LIN {X 0,Y 368.877,Z 478.526,A -85,B 0,C 180,E1 -12822.01,E2 -12822.01} C_VEL
LIN {X 0,Y 368.882,Z 478.53,A -85,B 0,C 180,E1 -12825.178,E2 -12825.178} C_VEL
LIN {X 0,Y 368.881,Z 478.519,A -85,B 0,C 180,E1 -12828.179,E2 -12828.179} C_VEL
LIN {X 0,Y 368.909,Z 478.528,A -85,B 0,C 180,E1 -12831.36,E2 -12831.36} C_VEL
LIN {X 0,Y 368.935,Z 478.472,A -85,B 0,C 180,E1 -12835.147,E2 -12835.147} C_VEL
LIN {X 0,Y 368.929,Z 478.53,A -85,B 0,C 180,E1 -12839.047,E2 -12839.047} C_VEL
LIN {X 0,Y 368.963,Z 478.492,A -85,B 0,C 180,E1 -12842.797,E2 -12842.797} C_VEL
LIN {X 0,Y 368.946,Z 478.523,A -85,B 0,C 180,E1 -12846.113,E2 -12846.113} C_VEL
LIN {X 0,Y 368.935,Z 478.655,A -85,B 0,C 180,E1 -12848.554,E2 -12848.554} C_VEL
LIN {X 0,Y 369.153,Z 479.57,A -85,B 0,C 180,E1 -12848.747,E2 -12848.747} C_VEL
LIN {X 0,Y 377.34,Z 498.899,A -85,B 0,C 180,E1 -12849.662,E2 -12849.662} C_VEL
LIN {X 0,Y 376.778,Z 559.865,A -85,B 0,C 180,E1 -12850.864,E2 -12850.864} C_VEL
LIN {X 0,Y 376.605,Z 573.144,A -85,B 0,C 180,E1 -12851.334,E2 -12851.334} C_VEL
LIN {X 0,Y 376.21,Z 585.351,A -85,B 0,C 180,E1 -12851.978,E2 -12851.978} C_VEL
LIN {X 0,Y 375.597,Z 597.68,A -85,B 0,C 180,E1 -12852.858,E2 -12852.858} C_VEL
LIN {X 0,Y 374.644,Z 609.255,A -85,B 0,C 180,E1 -12853.937,E2 -12853.937} C_VEL
LIN {X 0,Y 373.753,Z 619.585,A -85,B 0,C 180,E1 -12855.156,E2 -12855.156} C_VEL
LIN {X 0,Y 372.946,Z 628.011,A -85,B 0,C 180,E1 -12856.376,E2 -12856.376} C_VEL
LIN {X 0,Y 372.21,Z 635.75,A -85,B 0,C 180,E1 -12857.736,E2 -12857.736} C_VEL
LIN {X 0,Y 371.314,Z 643.431,A -85,B 0,C 180,E1 -12859.393,E2 -12859.393} C_VEL
LIN {X 0,Y 370.669,Z 649.183,A -85,B 0,C 180,E1 -12860.944,E2 -12860.944} C_VEL
LIN {X 0,Y 370.256,Z 653.452,A -85,B 0,C 180,E1 -12862.365,E2 -12862.365} C_VEL
LIN {X 0,Y 369.654,Z 657.346,A -85,B 0,C 180,E1 -12863.998,E2 -12863.998} C_VEL
LIN {X 0,Y 369.252,Z 660.212,A -85,B 0,C 180,E1 -12865.634,E2 -12865.634} C_VEL
LIN {X 0,Y 369.235,Z 661.562,A -85,B 0,C 180,E1 -12866.727,E2 -12866.727} C_VEL
LIN {X 0,Y 369.048,Z 662.545,A -85,B 0,C 180,E1 -12867.817,E2 -12867.817} C_VEL
LIN {X 0,Y 369.11,Z 663.126,A -85,B 0,C 180,E1 -12868.909,E2 -12868.909} C_VEL
LIN {X 0,Y 369.091,Z 663.354,A -85,B 0,C 180,E1 -12870,E2 -12870} C_VEL
LIN {X 0,Y 369.11,Z 663.169,A -85,B 0,C 180,E1 -12871.091,E2 -12871.091} C_VEL
LIN {X 0,Y 369.048,Z 662.615,A -85,B 0,C 180,E1 -12872.183,E2 -12872.183} C_VEL
LIN {X 0,Y 369.232,Z 661.661,A -85,B 0,C 180,E1 -12873.273,E2 -12873.273} C_VEL
LIN {X 0,Y 369.243,Z 660.356,A -85,B 0,C 180,E1 -12874.366,E2 -12874.366} C_VEL
LIN {X 0,Y 369.647,Z 657.542,A -85,B 0,C 180,E1 -12876.002,E2 -12876.002} C_VEL
LIN {X 0,Y 370.232,Z 653.717,A -85,B 0,C 180,E1 -12877.636,E2 -12877.636} C_VEL
LIN {X 0,Y 370.699,Z 648.641,A -85,B 0,C 180,E1 -12879.328,E2 -12879.328} C_VEL
LIN {X 0,Y 371.431,Z 642.614,A -85,B 0,C 180,E1 -12880.907,E2 -12880.907} C_VEL
LIN {X 0,Y 372.346,Z 634.835,A -85,B 0,C 180,E1 -12882.536,E2 -12882.536} C_VEL
LIN {X 0,Y 373.257,Z 625.165,A -85,B 0,C 180,E1 -12884.168,E2 -12884.168} C_VEL
LIN {X 0,Y 374.143,Z 616.123,A -85,B 0,C 180,E1 -12885.386,E2 -12885.386} C_VEL
LIN {X 0,Y 375.038,Z 605.628,A -85,B 0,C 180,E1 -12886.528,E2 -12886.528} C_VEL
LIN {X 0,Y 375.806,Z 593.96,A -85,B 0,C 180,E1 -12887.536,E2 -12887.536} C_VEL
LIN {X 0,Y 376.424,Z 582.268,A -85,B 0,C 180,E1 -12888.308,E2 -12888.308} C_VEL
LIN {X 0,Y 376.764,Z 569.639,A -85,B 0,C 180,E1 -12888.911,E2 -12888.911} C_VEL
LIN {X 0,Y 376.825,Z 558.831,A -85,B 0,C 180,E1 -12889.261,E2 -12889.261} C_VEL
LIN {X 0,Y 376.782,Z 552.259,A -85,B 0,C 180,E1 -12889.408,E2 -12889.408} C_VEL
LIN {X 0,Y 376.155,Z 546.467,A -85,B 0,C 180,E1 -12889.559,E2 -12889.559} C_VEL
LIN {X 0,Y 371.059,Z 527.828,A -85,B 0,C 180,E1 -12890.233,E2 -12890.233} C_VEL
LIN {X 0,Y 370.516,Z 522.033,A -85,B 0,C 180,E1 -12890.383,E2 -12890.383} C_VEL
LIN {X 0,Y 370.808,Z 500.919,A -85,B 0,C 180,E1 -12890.796,E2 -12890.796} C_VEL
LIN {X 0,Y 362.693,Z 481.915,A -85,B 0,C 180,E1 -12891.708,E2 -12891.708} C_VEL
LIN {X 0,Y 361.991,Z 479.937,A -85,B 0,C 180,E1 -12891.87,E2 -12891.87} C_VEL
LIN {X 0,Y 361.91,Z 479.438,A -85,B 0,C 180,E1 -12892.1,E2 -12892.1} C_VEL
LIN {X 0,Y 361.929,Z 479.391,A -85,B 0,C 180,E1 -12895.289,E2 -12895.289} C_VEL
LIN {X 0,Y 361.908,Z 479.371,A -85,B 0,C 180,E1 -12897.778,E2 -12897.778} C_VEL
LIN {X 0,Y 361.837,Z 479.406,A -85,B 0,C 180,E1 -12901.629,E2 -12901.629} C_VEL
LIN {X 0,Y 361.873,Z 479.404,A -85,B 0,C 180,E1 -12905.344,E2 -12905.344} C_VEL
LIN {X 0,Y 361.869,Z 479.409,A -85,B 0,C 180,E1 -12909.026,E2 -12909.026} C_VEL
LIN {X 0,Y 361.833,Z 479.393,A -85,B 0,C 180,E1 -12912.828,E2 -12912.828} C_VEL
LIN {X 0,Y 361.832,Z 479.413,A -85,B 0,C 180,E1 -12915.943,E2 -12915.943} C_VEL
LIN {X 0,Y 361.83,Z 479.384,A -85,B 0,C 180,E1 -12919.244,E2 -12919.244} C_VEL
LIN {X 0,Y 361.859,Z 479.402,A -85,B 0,C 180,E1 -12922.776,E2 -12922.776} C_VEL
LIN {X 0,Y 361.849,Z 479.405,A -85,B 0,C 180,E1 -12925.719,E2 -12925.719} C_VEL
LIN {X 0,Y 361.871,Z 479.368,A -85,B 0,C 180,E1 -12929.672,E2 -12929.672} C_VEL
LIN {X 0,Y 361.949,Z 479.398,A -85,B 0,C 180,E1 -12933.474,E2 -12933.474} C_VEL
LIN {X 0,Y 361.883,Z 479.398,A -85,B 0,C 180,E1 -12937.144,E2 -12937.144} C_VEL
LIN {X 0,Y 361.899,Z 479.404,A -85,B 0,C 180,E1 -12940.723,E2 -12940.723} C_VEL
LIN {X 0,Y 361.925,Z 479.393,A -85,B 0,C 180,E1 -12943.066,E2 -12943.066} C_VEL
LIN {X 0,Y 361.991,Z 479.391,A -85,B 0,C 180,E1 -12946.527,E2 -12946.527} C_VEL
LIN {X 0,Y 362.024,Z 479.374,A -85,B 0,C 180,E1 -12949.938,E2 -12949.938} C_VEL
LIN {X 0,Y 362.143,Z 479.368,A -85,B 0,C 180,E1 -12952.192,E2 -12952.192} C_VEL
LIN {X 0,Y 362.11,Z 479.374,A -85,B 0,C 180,E1 -12954.431,E2 -12954.431} C_VEL
LIN {X 0,Y 362.275,Z 479.344,A -85,B 0,C 180,E1 -12957.776,E2 -12957.776} C_VEL
LIN {X 0,Y 362.421,Z 479.336,A -85,B 0,C 180,E1 -12960,E2 -12960} C_VEL
LIN {X 0,Y 362.275,Z 479.35,A -85,B 0,C 180,E1 -12962.224,E2 -12962.224} C_VEL
LIN {X 0,Y 362.16,Z 479.368,A -85,B 0,C 180,E1 -12966.686,E2 -12966.686} C_VEL
LIN {X 0,Y 362.023,Z 479.377,A -85,B 0,C 180,E1 -12970.062,E2 -12970.062} C_VEL
LIN {X 0,Y 361.99,Z 479.394,A -85,B 0,C 180,E1 -12973.899,E2 -12973.899} C_VEL
LIN {X 0,Y 361.96,Z 479.372,A -85,B 0,C 180,E1 -12977.939,E2 -12977.939} C_VEL
LIN {X 0,Y 361.876,Z 479.403,A -85,B 0,C 180,E1 -12981.654,E2 -12981.654} C_VEL
LIN {X 0,Y 361.921,Z 479.393,A -85,B 0,C 180,E1 -12985.291,E2 -12985.291} C_VEL
LIN {X 0,Y 361.917,Z 479.387,A -85,B 0,C 180,E1 -12987.778,E2 -12987.778} C_VEL
LIN {X 0,Y 361.841,Z 479.413,A -85,B 0,C 180,E1 -12991.286,E2 -12991.286} C_VEL
LIN {X 0,Y 361.849,Z 479.406,A -85,B 0,C 180,E1 -12994.281,E2 -12994.281} C_VEL
LIN {X 0,Y 361.86,Z 479.407,A -85,B 0,C 180,E1 -12997.224,E2 -12997.224} C_VEL
LIN {X 0,Y 361.832,Z 479.413,A -85,B 0,C 180,E1 -13000.756,E2 -13000.756} C_VEL
LIN {X 0,Y 361.842,Z 479.382,A -85,B 0,C 180,E1 -13004.365,E2 -13004.365} C_VEL
LIN {X 0,Y 361.881,Z 479.408,A -85,B 0,C 180,E1 -13007.561,E2 -13007.561} C_VEL
LIN {X 0,Y 361.872,Z 479.401,A -85,B 0,C 180,E1 -13010.973,E2 -13010.973} C_VEL
LIN {X 0,Y 361.906,Z 479.544,A -85,B 0,C 180,E1 -13014.756,E2 -13014.756} C_VEL
LIN {X 0,Y 365.118,Z 492.779,A -85,B 0,C 180,E1 -13017.591,E2 -13017.591} C_VEL
LIN {X 0,Y 367.943,Z 505.89,A -85,B 0,C 180,E1 -13020.224,E2 -13020.224} C_VEL
LIN {X 0,Y 367.28,Z 514.74,A -85,B 0,C 180,E1 -13021.796,E2 -13021.796} C_VEL
LIN {X 0,Y 364.961,Z 539.488,A -85,B 0,C 180,E1 -13026.148,E2 -13026.148} C_VEL
LIN {X 0,Y 364.188,Z 549.23,A -85,B 0,C 180,E1 -13027.834,E2 -13027.834} C_VEL
LIN {X 0,Y 368.3,Z 584.784,A -85,B 0,C 180,E1 -13028.832,E2 -13028.832} C_VEL
LIN {X 0,Y 369.534,Z 599.506,A -85,B 0,C 180,E1 -13029.201,E2 -13029.201} C_VEL
LIN {X 0,Y 368.537,Z 660.016,A -85,B 0,C 180,E1 -13030.397,E2 -13030.397} C_VEL
LIN {X 0,Y 367.865,Z 673.29,A -85,B 0,C 180,E1 -13030.867,E2 -13030.867} C_VEL
LIN {X 0,Y 366.915,Z 685.485,A -85,B 0,C 180,E1 -13031.504,E2 -13031.504} C_VEL
LIN {X 0,Y 365.68,Z 697.816,A -85,B 0,C 180,E1 -13032.381,E2 -13032.381} C_VEL
LIN {X 0,Y 364.603,Z 709.538,A -85,B 0,C 180,E1 -13033.482,E2 -13033.482} C_VEL
LIN {X 0,Y 363.558,Z 719.018,A -85,B 0,C 180,E1 -13034.586,E2 -13034.586} C_VEL
LIN {X 0,Y 362.501,Z 728.498,A -85,B 0,C 180,E1 -13035.932,E2 -13035.932} C_VEL
LIN {X 0,Y 362.19,Z 733.797,A -85,B 0,C 180,E1 -13036.821,E2 -13036.821} C_VEL
LIN {X 0,Y 361.524,Z 740.995,A -85,B 0,C 180,E1 -13038.222,E2 -13038.222} C_VEL
LIN {X 0,Y 361.08,Z 748.089,A -85,B 0,C 180,E1 -13039.911,E2 -13039.911} C_VEL
LIN {X 0,Y 360.92,Z 753.811,A -85,B 0,C 180,E1 -13041.603,E2 -13041.603} C_VEL
LIN {X 0,Y 360.946,Z 758.327,A -85,B 0,C 180,E1 -13043.291,E2 -13043.291} C_VEL
LIN {X 0,Y 361.025,Z 760.727,A -85,B 0,C 180,E1 -13044.414,E2 -13044.414} C_VEL
LIN {X 0,Y 361.182,Z 762.687,A -85,B 0,C 180,E1 -13045.536,E2 -13045.536} C_VEL
LIN {X 0,Y 361.271,Z 764.153,A -85,B 0,C 180,E1 -13046.654,E2 -13046.654} C_VEL
LIN {X 0,Y 361.67,Z 765.879,A -85,B 0,C 180,E1 -13048.887,E2 -13048.887} C_VEL
LIN {X 0,Y 361.734,Z 766.112,A -85,B 0,C 180,E1 -13050,E2 -13050} C_VEL
LIN {X 0,Y 361.67,Z 765.876,A -85,B 0,C 180,E1 -13051.113,E2 -13051.113} C_VEL
LIN {X 0,Y 361.274,Z 764.148,A -85,B 0,C 180,E1 -13053.346,E2 -13053.346} C_VEL
LIN {X 0,Y 361.19,Z 762.678,A -85,B 0,C 180,E1 -13054.464,E2 -13054.464} C_VEL
LIN {X 0,Y 361.019,Z 759.595,A -85,B 0,C 180,E1 -13056.146,E2 -13056.146} C_VEL
LIN {X 0,Y 360.914,Z 755.441,A -85,B 0,C 180,E1 -13057.834,E2 -13057.834} C_VEL
LIN {X 0,Y 361.055,Z 749.1,A -85,B 0,C 180,E1 -13059.806,E2 -13059.806} C_VEL
LIN {X 0,Y 361.453,Z 742.222,A -85,B 0,C 180,E1 -13061.496,E2 -13061.496} C_VEL
LIN {X 0,Y 362.184,Z 733.742,A -85,B 0,C 180,E1 -13063.179,E2 -13063.179} C_VEL
LIN {X 0,Y 362.895,Z 725.06,A -85,B 0,C 180,E1 -13064.582,E2 -13064.582} C_VEL
LIN {X 0,Y 363.82,Z 715.587,A -85,B 0,C 180,E1 -13065.834,E2 -13065.834} C_VEL
LIN {X 0,Y 365.095,Z 703.902,A -85,B 0,C 180,E1 -13067.071,E2 -13067.071} C_VEL
LIN {X 0,Y 366.265,Z 692.423,A -85,B 0,C 180,E1 -13068.023,E2 -13068.023} C_VEL
LIN {X 0,Y 367.281,Z 680.646,A -85,B 0,C 180,E1 -13068.766,E2 -13068.766} C_VEL
LIN {X 0,Y 368.186,Z 667.106,A -85,B 0,C 180,E1 -13069.369,E2 -13069.369} C_VEL
LIN {X 0,Y 368.651,Z 653.646,A -85,B 0,C 180,E1 -13069.742,E2 -13069.742} C_VEL
LIN {X 0,Y 369.378,Z 596.606,A -85,B 0,C 180,E1 -13070.854,E2 -13070.854} C_VEL
LIN {X 0,Y 365.691,Z 561.697,A -85,B 0,C 180,E1 -13071.779,E2 -13071.779} C_VEL
LIN {X 0,Y 364.181,Z 549.137,A -85,B 0,C 180,E1 -13072.162,E2 -13072.162} C_VEL
LIN {X 0,Y 366.138,Z 526.073,A -85,B 0,C 180,E1 -13076.198,E2 -13076.198} C_VEL
LIN {X 0,Y 367.987,Z 507.54,A -85,B 0,C 180,E1 -13079.457,E2 -13079.457} C_VEL
LIN {X 0,Y 367.443,Z 503.107,A -85,B 0,C 180,E1 -13080.304,E2 -13080.304} C_VEL
LIN {X 0,Y 363.861,Z 487.384,A -85,B 0,C 180,E1 -13083.515,E2 -13083.515} C_VEL
LIN {X 0,Y 361.898,Z 479.519,A -85,B 0,C 180,E1 -13085.245,E2 -13085.245} C_VEL
LIN {X 0,Y 361.872,Z 479.401,A -85,B 0,C 180,E1 -13089.027,E2 -13089.027} C_VEL
LIN {X 0,Y 361.881,Z 479.409,A -85,B 0,C 180,E1 -13092.439,E2 -13092.439} C_VEL
LIN {X 0,Y 361.842,Z 479.382,A -85,B 0,C 180,E1 -13095.635,E2 -13095.635} C_VEL
LIN {X 0,Y 361.832,Z 479.412,A -85,B 0,C 180,E1 -13099.244,E2 -13099.244} C_VEL
LIN {X 0,Y 361.86,Z 479.407,A -85,B 0,C 180,E1 -13102.776,E2 -13102.776} C_VEL
LIN {X 0,Y 361.849,Z 479.405,A -85,B 0,C 180,E1 -13105.719,E2 -13105.719} C_VEL
LIN {X 0,Y 361.872,Z 479.408,A -85,B 0,C 180,E1 -13109.672,E2 -13109.672} C_VEL
LIN {X 0,Y 361.948,Z 479.378,A -85,B 0,C 180,E1 -13113.475,E2 -13113.475} C_VEL
LIN {X 0,Y 361.883,Z 479.405,A -85,B 0,C 180,E1 -13117.144,E2 -13117.144} C_VEL
LIN {X 0,Y 361.881,Z 479.38,A -85,B 0,C 180,E1 -13120.722,E2 -13120.722} C_VEL
LIN {X 0,Y 361.925,Z 479.393,A -85,B 0,C 180,E1 -13123.066,E2 -13123.066} C_VEL
LIN {X 0,Y 361.991,Z 479.393,A -85,B 0,C 180,E1 -13126.528,E2 -13126.528} C_VEL
LIN {X 0,Y 362.023,Z 479.378,A -85,B 0,C 180,E1 -13129.938,E2 -13129.938} C_VEL
LIN {X 0,Y 362.16,Z 479.368,A -85,B 0,C 180,E1 -13133.314,E2 -13133.314} C_VEL
LIN {X 0,Y 362.275,Z 479.353,A -85,B 0,C 180,E1 -13137.776,E2 -13137.776} C_VEL
LIN {X 0,Y 362.421,Z 479.338,A -85,B 0,C 180,E1 -13140,E2 -13140} C_VEL
LIN {X 0,Y 362.275,Z 479.346,A -85,B 0,C 180,E1 -13142.224,E2 -13142.224} C_VEL
LIN {X 0,Y 362.16,Z 479.372,A -85,B 0,C 180,E1 -13146.686,E2 -13146.686} C_VEL
LIN {X 0,Y 362.024,Z 479.374,A -85,B 0,C 180,E1 -13150.062,E2 -13150.062} C_VEL
LIN {X 0,Y 361.99,Z 479.39,A -85,B 0,C 180,E1 -13153.899,E2 -13153.899} C_VEL
LIN {X 0,Y 361.96,Z 479.392,A -85,B 0,C 180,E1 -13157.939,E2 -13157.939} C_VEL
LIN {X 0,Y 361.876,Z 479.397,A -85,B 0,C 180,E1 -13161.654,E2 -13161.654} C_VEL
LIN {X 0,Y 361.922,Z 479.402,A -85,B 0,C 180,E1 -13165.291,E2 -13165.291} C_VEL
LIN {X 0,Y 361.916,Z 479.391,A -85,B 0,C 180,E1 -13167.779,E2 -13167.779} C_VEL
LIN {X 0,Y 361.841,Z 479.373,A -85,B 0,C 180,E1 -13171.286,E2 -13171.286} C_VEL
LIN {X 0,Y 361.849,Z 479.404,A -85,B 0,C 180,E1 -13174.281,E2 -13174.281} C_VEL
LIN {X 0,Y 361.859,Z 479.403,A -85,B 0,C 180,E1 -13177.224,E2 -13177.224} C_VEL
LIN {X 0,Y 361.83,Z 479.384,A -85,B 0,C 180,E1 -13180.756,E2 -13180.756} C_VEL
LIN {X 0,Y 361.843,Z 479.412,A -85,B 0,C 180,E1 -13184.365,E2 -13184.365} C_VEL
LIN {X 0,Y 361.834,Z 479.392,A -85,B 0,C 180,E1 -13187.569,E2 -13187.569} C_VEL
LIN {X 0,Y 361.87,Z 479.409,A -85,B 0,C 180,E1 -13190.974,E2 -13190.974} C_VEL
LIN {X 0,Y 361.873,Z 479.354,A -85,B 0,C 180,E1 -13194.656,E2 -13194.656} C_VEL
LIN {X 0,Y 361.837,Z 479.405,A -85,B 0,C 180,E1 -13198.371,E2 -13198.371} C_VEL
LIN {X 0,Y 361.908,Z 479.373,A -85,B 0,C 180,E1 -13202.222,E2 -13202.222} C_VEL
LIN {X 0,Y 361.929,Z 479.389,A -85,B 0,C 180,E1 -13204.711,E2 -13204.711} C_VEL
LIN {X 0,Y 361.913,Z 479.54,A -85,B 0,C 180,E1 -13208.124,E2 -13208.124} C_VEL
LIN {X 0,Y 362.139,Z 480.575,A -85,B 0,C 180,E1 -13208.317,E2 -13208.317} C_VEL
LIN {X 0,Y 370.357,Z 499.721,A -85,B 0,C 180,E1 -13209.256,E2 -13209.256} C_VEL
LIN {X 0,Y 370.821,Z 501.605,A -85,B 0,C 180,E1 -13209.323,E2 -13209.323} C_VEL
LIN {X 0,Y 370.139,Z 559.915,A -85,B 0,C 180,E1 -13210.484,E2 -13210.484} C_VEL
LIN {X 0,Y 369.975,Z 572.765,A -85,B 0,C 180,E1 -13210.921,E2 -13210.921} C_VEL
LIN {X 0,Y 369.575,Z 585.231,A -85,B 0,C 180,E1 -13211.571,E2 -13211.571} C_VEL
LIN {X 0,Y 368.939,Z 597.581,A -85,B 0,C 180,E1 -13212.448,E2 -13212.448} C_VEL
LIN {X 0,Y 368.008,Z 608.977,A -85,B 0,C 180,E1 -13213.497,E2 -13213.497} C_VEL
LIN {X 0,Y 367.031,Z 619.532,A -85,B 0,C 180,E1 -13214.735,E2 -13214.735} C_VEL
LIN {X 0,Y 366.119,Z 629.002,A -85,B 0,C 180,E1 -13216.117,E2 -13216.117} C_VEL
LIN {X 0,Y 365.345,Z 636.74,A -85,B 0,C 180,E1 -13217.502,E2 -13217.502} C_VEL
LIN {X 0,Y 364.409,Z 644.421,A -85,B 0,C 180,E1 -13219.19,E2 -13219.19} C_VEL
LIN {X 0,Y 363.73,Z 650.173,A -85,B 0,C 180,E1 -13220.77,E2 -13220.77} C_VEL
LIN {X 0,Y 363.292,Z 654.441,A -85,B 0,C 180,E1 -13222.217,E2 -13222.217} C_VEL
LIN {X 0,Y 362.665,Z 658.335,A -85,B 0,C 180,E1 -13223.882,E2 -13223.882} C_VEL
LIN {X 0,Y 362.243,Z 661.202,A -85,B 0,C 180,E1 -13225.549,E2 -13225.549} C_VEL
LIN {X 0,Y 362.218,Z 662.551,A -85,B 0,C 180,E1 -13226.663,E2 -13226.663} C_VEL
LIN {X 0,Y 362.027,Z 663.533,A -85,B 0,C 180,E1 -13227.775,E2 -13227.775} C_VEL
LIN {X 0,Y 362.085,Z 664.114,A -85,B 0,C 180,E1 -13228.888,E2 -13228.888} C_VEL
LIN {X 0,Y 362.065,Z 664.342,A -85,B 0,C 180,E1 -13230,E2 -13230} C_VEL
LIN {X 0,Y 362.085,Z 664.156,A -85,B 0,C 180,E1 -13231.112,E2 -13231.112} C_VEL
LIN {X 0,Y 362.026,Z 663.603,A -85,B 0,C 180,E1 -13232.225,E2 -13232.225} C_VEL
LIN {X 0,Y 362.215,Z 662.648,A -85,B 0,C 180,E1 -13233.337,E2 -13233.337} C_VEL
LIN {X 0,Y 362.232,Z 661.344,A -85,B 0,C 180,E1 -13234.451,E2 -13234.451} C_VEL
LIN {X 0,Y 362.657,Z 658.53,A -85,B 0,C 180,E1 -13236.118,E2 -13236.118} C_VEL
LIN {X 0,Y 363.268,Z 654.704,A -85,B 0,C 180,E1 -13237.783,E2 -13237.783} C_VEL
LIN {X 0,Y 363.765,Z 649.628,A -85,B 0,C 180,E1 -13239.508,E2 -13239.508} C_VEL
LIN {X 0,Y 364.532,Z 643.6,A -85,B 0,C 180,E1 -13241.116,E2 -13241.116} C_VEL
LIN {X 0,Y 365.488,Z 635.821,A -85,B 0,C 180,E1 -13242.775,E2 -13242.775} C_VEL
LIN {X 0,Y 366.445,Z 626.151,A -85,B 0,C 180,E1 -13244.437,E2 -13244.437} C_VEL
LIN {X 0,Y 367.355,Z 617.11,A -85,B 0,C 180,E1 -13245.678,E2 -13245.678} C_VEL
LIN {X 0,Y 368.301,Z 606.613,A -85,B 0,C 180,E1 -13246.839,E2 -13246.839} C_VEL
LIN {X 0,Y 369.089,Z 595.098,A -85,B 0,C 180,E1 -13247.853,E2 -13247.853} C_VEL
LIN {X 0,Y 369.752,Z 583.832,A -85,B 0,C 180,E1 -13248.614,E2 -13248.614} C_VEL
LIN {X 0,Y 370.09,Z 571.524,A -85,B 0,C 180,E1 -13249.229,E2 -13249.229} C_VEL
LIN {X 0,Y 370.196,Z 559.798,A -85,B 0,C 180,E1 -13249.62,E2 -13249.62} C_VEL
LIN {X 0,Y 370.506,Z 523.206,A -85,B 0,C 180,E1 -13250.36,E2 -13250.36} C_VEL
LIN {X 0,Y 370.516,Z 522.033,A -85,B 0,C 180,E1 -13250.383,E2 -13250.383} C_VEL
LIN {X 0,Y 369.893,Z 516.227,A -85,B 0,C 180,E1 -13250.54,E2 -13250.54} C_VEL
LIN {X 0,Y 368.235,Z 510.668,A -85,B 0,C 180,E1 -13250.756,E2 -13250.756} C_VEL
LIN {X 0,Y 360.193,Z 492.917,A -85,B 0,C 180,E1 -13251.641,E2 -13251.641} C_VEL
LIN {X 0,Y 355.081,Z 481.33,A -85,B 0,C 180,E1 -13252.256,E2 -13252.256} C_VEL
LIN {X 0,Y 354.878,Z 480.41,A -85,B 0,C 180,E1 -13252.462,E2 -13252.462} C_VEL
LIN {X 0,Y 354.9,Z 480.253,A -85,B 0,C 180,E1 -13255.827,E2 -13255.827} C_VEL
LIN {X 0,Y 354.817,Z 480.284,A -85,B 0,C 180,E1 -13259.681,E2 -13259.681} C_VEL
LIN {X 0,Y 354.805,Z 480.288,A -85,B 0,C 180,E1 -13263.701,E2 -13263.701} C_VEL
LIN {X 0,Y 354.797,Z 480.277,A -85,B 0,C 180,E1 -13266.459,E2 -13266.459} C_VEL
LIN {X 0,Y 354.822,Z 480.289,A -85,B 0,C 180,E1 -13269.423,E2 -13269.423} C_VEL
LIN {X 0,Y 354.785,Z 480.27,A -85,B 0,C 180,E1 -13272.866,E2 -13272.866} C_VEL
LIN {X 0,Y 354.778,Z 480.292,A -85,B 0,C 180,E1 -13276.105,E2 -13276.105} C_VEL
LIN {X 0,Y 354.783,Z 480.262,A -85,B 0,C 180,E1 -13279.178,E2 -13279.178} C_VEL
LIN {X 0,Y 354.803,Z 480.279,A -85,B 0,C 180,E1 -13282.402,E2 -13282.402} C_VEL
LIN {X 0,Y 354.808,Z 480.291,A -85,B 0,C 180,E1 -13284.94,E2 -13284.94} C_VEL
LIN {X 0,Y 354.788,Z 480.254,A -85,B 0,C 180,E1 -13288.404,E2 -13288.404} C_VEL
LIN {X 0,Y 354.848,Z 480.263,A -85,B 0,C 180,E1 -13291.619,E2 -13291.619} C_VEL
LIN {X 0,Y 354.893,Z 480.275,A -85,B 0,C 180,E1 -13294.172,E2 -13294.172} C_VEL
LIN {X 0,Y 354.823,Z 480.275,A -85,B 0,C 180,E1 -13297.893,E2 -13297.893} C_VEL
LIN {X 0,Y 354.915,Z 480.27,A -85,B 0,C 180,E1 -13301.891,E2 -13301.891} C_VEL
LIN {X 0,Y 354.935,Z 480.27,A -85,B 0,C 180,E1 -13305.981,E2 -13305.981} C_VEL
LIN {X 0,Y 354.97,Z 480.253,A -85,B 0,C 180,E1 -13309.736,E2 -13309.736} C_VEL
LIN {X 0,Y 355.106,Z 480.245,A -85,B 0,C 180,E1 -13312.037,E2 -13312.037} C_VEL
LIN {X 0,Y 355.084,Z 480.249,A -85,B 0,C 180,E1 -13314.32,E2 -13314.32} C_VEL
LIN {X 0,Y 355.238,Z 480.22,A -85,B 0,C 180,E1 -13317.732,E2 -13317.732} C_VEL
LIN {X 0,Y 355.391,Z 480.212,A -85,B 0,C 180,E1 -13320,E2 -13320} C_VEL
LIN {X 0,Y 355.238,Z 480.226,A -85,B 0,C 180,E1 -13322.268,E2 -13322.268} C_VEL
LIN {X 0,Y 355.122,Z 480.245,A -85,B 0,C 180,E1 -13326.819,E2 -13326.819} C_VEL
LIN {X 0,Y 354.97,Z 480.254,A -85,B 0,C 180,E1 -13330.264,E2 -13330.264} C_VEL
LIN {X 0,Y 354.935,Z 480.272,A -85,B 0,C 180,E1 -13334.019,E2 -13334.019} C_VEL
LIN {X 0,Y 354.915,Z 480.248,A -85,B 0,C 180,E1 -13338.109,E2 -13338.109} C_VEL
LIN {X 0,Y 354.823,Z 480.286,A -85,B 0,C 180,E1 -13342.107,E2 -13342.107} C_VEL
LIN {X 0,Y 354.893,Z 480.26,A -85,B 0,C 180,E1 -13345.828,E2 -13345.828} C_VEL
LIN {X 0,Y 354.849,Z 480.284,A -85,B 0,C 180,E1 -13349.679,E2 -13349.679} C_VEL
LIN {X 0,Y 354.801,Z 480.276,A -85,B 0,C 180,E1 -13353.703,E2 -13353.703} C_VEL
LIN {X 0,Y 354.793,Z 480.288,A -85,B 0,C 180,E1 -13356.46,E2 -13356.46} C_VEL
LIN {X 0,Y 354.82,Z 480.283,A -85,B 0,C 180,E1 -13359.424,E2 -13359.424} C_VEL
LIN {X 0,Y 354.786,Z 480.268,A -85,B 0,C 180,E1 -13362.868,E2 -13362.868} C_VEL
LIN {X 0,Y 354.849,Z 480.277,A -85,B 0,C 180,E1 -13366.118,E2 -13366.118} C_VEL
LIN {X 0,Y 354.853,Z 480.264,A -85,B 0,C 180,E1 -13369.189,E2 -13369.189} C_VEL
LIN {X 0,Y 354.807,Z 480.284,A -85,B 0,C 180,E1 -13372.403,E2 -13372.403} C_VEL
LIN {X 0,Y 354.863,Z 480.538,A -85,B 0,C 180,E1 -13374.363,E2 -13374.363} C_VEL
LIN {X 0,Y 358.004,Z 493.339,A -85,B 0,C 180,E1 -13377.169,E2 -13377.169} C_VEL
LIN {X 0,Y 360.932,Z 506.614,A -85,B 0,C 180,E1 -13379.908,E2 -13379.908} C_VEL
LIN {X 0,Y 360.973,Z 510.056,A -85,B 0,C 180,E1 -13380.555,E2 -13380.555} C_VEL
LIN {X 0,Y 358.83,Z 530.823,A -85,B 0,C 180,E1 -13384.284,E2 -13384.284} C_VEL
LIN {X 0,Y 357.342,Z 548.301,A -85,B 0,C 180,E1 -13387.392,E2 -13387.392} C_VEL
LIN {X 0,Y 361.535,Z 584.354,A -85,B 0,C 180,E1 -13388.428,E2 -13388.428} C_VEL
LIN {X 0,Y 362.817,Z 600.626,A -85,B 0,C 180,E1 -13388.841,E2 -13388.841} C_VEL
LIN {X 0,Y 361.821,Z 659.025,A -85,B 0,C 180,E1 -13390.018,E2 -13390.018} C_VEL
LIN {X 0,Y 361.137,Z 672.296,A -85,B 0,C 180,E1 -13390.496,E2 -13390.496} C_VEL
LIN {X 0,Y 360.142,Z 684.486,A -85,B 0,C 180,E1 -13391.143,E2 -13391.143} C_VEL
LIN {X 0,Y 358.907,Z 696.821,A -85,B 0,C 180,E1 -13392.037,E2 -13392.037} C_VEL
LIN {X 0,Y 357.72,Z 708.531,A -85,B 0,C 180,E1 -13393.155,E2 -13393.155} C_VEL
LIN {X 0,Y 356.643,Z 718.012,A -85,B 0,C 180,E1 -13394.279,E2 -13394.279} C_VEL
LIN {X 0,Y 355.627,Z 726.828,A -85,B 0,C 180,E1 -13395.548,E2 -13395.548} C_VEL
LIN {X 0,Y 355.032,Z 734.309,A -85,B 0,C 180,E1 -13396.842,E2 -13396.842} C_VEL
LIN {X 0,Y 354.324,Z 742.526,A -85,B 0,C 180,E1 -13398.56,E2 -13398.56} C_VEL
LIN {X 0,Y 353.955,Z 749.161,A -85,B 0,C 180,E1 -13400.284,E2 -13400.284} C_VEL
LIN {X 0,Y 353.843,Z 754.464,A -85,B 0,C 180,E1 -13402.008,E2 -13402.008} C_VEL
LIN {X 0,Y 353.909,Z 758.206,A -85,B 0,C 180,E1 -13403.543,E2 -13403.543} C_VEL
LIN {X 0,Y 354.119,Z 761.691,A -85,B 0,C 180,E1 -13405.447,E2 -13405.447} C_VEL
LIN {X 0,Y 354.221,Z 763.161,A -85,B 0,C 180,E1 -13406.588,E2 -13406.588} C_VEL
LIN {X 0,Y 354.637,Z 764.89,A -85,B 0,C 180,E1 -13408.864,E2 -13408.864} C_VEL
LIN {X 0,Y 354.709,Z 765.124,A -85,B 0,C 180,E1 -13410,E2 -13410} C_VEL
LIN {X 0,Y 354.637,Z 764.887,A -85,B 0,C 180,E1 -13411.136,E2 -13411.136} C_VEL
LIN {X 0,Y 354.225,Z 763.155,A -85,B 0,C 180,E1 -13413.412,E2 -13413.412} C_VEL
LIN {X 0,Y 354.125,Z 761.681,A -85,B 0,C 180,E1 -13414.553,E2 -13414.553} C_VEL
LIN {X 0,Y 353.92,Z 758.147,A -85,B 0,C 180,E1 -13416.474,E2 -13416.474} C_VEL
LIN {X 0,Y 353.867,Z 752.778,A -85,B 0,C 180,E1 -13418.566,E2 -13418.566} C_VEL
LIN {X 0,Y 354.011,Z 747.043,A -85,B 0,C 180,E1 -13420.292,E2 -13420.292} C_VEL
LIN {X 0,Y 354.52,Z 739.942,A -85,B 0,C 180,E1 -13422.014,E2 -13422.014} C_VEL
LIN {X 0,Y 355.241,Z 732.737,A -85,B 0,C 180,E1 -13423.442,E2 -13423.442} C_VEL
LIN {X 0,Y 355.982,Z 724.052,A -85,B 0,C 180,E1 -13424.871,E2 -13424.871} C_VEL
LIN {X 0,Y 356.917,Z 714.574,A -85,B 0,C 180,E1 -13426.148,E2 -13426.148} C_VEL
LIN {X 0,Y 358.292,Z 702.896,A -85,B 0,C 180,E1 -13427.405,E2 -13427.405} C_VEL
LIN {X 0,Y 359.506,Z 691.418,A -85,B 0,C 180,E1 -13428.374,E2 -13428.374} C_VEL
LIN {X 0,Y 360.558,Z 679.639,A -85,B 0,C 180,E1 -13429.129,E2 -13429.129} C_VEL
LIN {X 0,Y 361.478,Z 666.094,A -85,B 0,C 180,E1 -13429.743,E2 -13429.743} C_VEL
LIN {X 0,Y 361.97,Z 652.626,A -85,B 0,C 180,E1 -13430.122,E2 -13430.122} C_VEL
LIN {X 0,Y 362.718,Z 597.263,A -85,B 0,C 180,E1 -13431.221,E2 -13431.221} C_VEL
LIN {X 0,Y 358.867,Z 560.876,A -85,B 0,C 180,E1 -13432.211,E2 -13432.211} C_VEL
LIN {X 0,Y 357.321,Z 548.227,A -85,B 0,C 180,E1 -13432.599,E2 -13432.599} C_VEL
LIN {X 0,Y 359.245,Z 526.704,A -85,B 0,C 180,E1 -13436.437,E2 -13436.437} C_VEL
LIN {X 0,Y 361.115,Z 508.278,A -85,B 0,C 180,E1 -13439.753,E2 -13439.753} C_VEL
LIN {X 0,Y 359.378,Z 499.232,A -85,B 0,C 180,E1 -13441.576,E2 -13441.576} C_VEL
LIN {X 0,Y 355.943,Z 484.627,A -85,B 0,C 180,E1 -13444.685,E2 -13444.685} C_VEL
LIN {X 0,Y 354.837,Z 480.365,A -85,B 0,C 180,E1 -13445.702,E2 -13445.702} C_VEL
LIN {X 0,Y 354.821,Z 480.272,A -85,B 0,C 180,E1 -13449.423,E2 -13449.423} C_VEL
LIN {X 0,Y 354.832,Z 480.288,A -85,B 0,C 180,E1 -13452.875,E2 -13452.875} C_VEL
LIN {X 0,Y 354.779,Z 480.26,A -85,B 0,C 180,E1 -13456.105,E2 -13456.105} C_VEL
LIN {X 0,Y 354.784,Z 480.29,A -85,B 0,C 180,E1 -13459.178,E2 -13459.178} C_VEL
LIN {X 0,Y 354.803,Z 480.281,A -85,B 0,C 180,E1 -13462.402,E2 -13462.402} C_VEL
LIN {X 0,Y 354.807,Z 480.285,A -85,B 0,C 180,E1 -13464.94,E2 -13464.94} C_VEL
LIN {X 0,Y 354.788,Z 480.287,A -85,B 0,C 180,E1 -13468.404,E2 -13468.404} C_VEL
LIN {X 0,Y 354.849,Z 480.276,A -85,B 0,C 180,E1 -13471.619,E2 -13471.619} C_VEL
LIN {X 0,Y 354.893,Z 480.261,A -85,B 0,C 180,E1 -13474.172,E2 -13474.172} C_VEL
LIN {X 0,Y 354.823,Z 480.285,A -85,B 0,C 180,E1 -13477.893,E2 -13477.893} C_VEL
LIN {X 0,Y 354.915,Z 480.249,A -85,B 0,C 180,E1 -13481.891,E2 -13481.891} C_VEL
LIN {X 0,Y 354.935,Z 480.272,A -85,B 0,C 180,E1 -13485.981,E2 -13485.981} C_VEL
LIN {X 0,Y 354.97,Z 480.256,A -85,B 0,C 180,E1 -13489.736,E2 -13489.736} C_VEL
LIN {X 0,Y 355.122,Z 480.246,A -85,B 0,C 180,E1 -13493.181,E2 -13493.181} C_VEL
LIN {X 0,Y 355.238,Z 480.229,A -85,B 0,C 180,E1 -13497.732,E2 -13497.732} C_VEL
LIN {X 0,Y 355.391,Z 480.214,A -85,B 0,C 180,E1 -13500,E2 -13500} C_VEL
LIN {X 0,Y 355.238,Z 480.222,A -85,B 0,C 180,E1 -13502.268,E2 -13502.268} C_VEL
LIN {X 0,Y 355.122,Z 480.247,A -85,B 0,C 180,E1 -13506.82,E2 -13506.82} C_VEL
LIN {X 0,Y 354.97,Z 480.253,A -85,B 0,C 180,E1 -13510.264,E2 -13510.264} C_VEL
LIN {X 0,Y 354.935,Z 480.27,A -85,B 0,C 180,E1 -13514.019,E2 -13514.019} C_VEL
LIN {X 0,Y 354.915,Z 480.27,A -85,B 0,C 180,E1 -13518.109,E2 -13518.109} C_VEL
LIN {X 0,Y 354.823,Z 480.275,A -85,B 0,C 180,E1 -13522.107,E2 -13522.107} C_VEL
LIN {X 0,Y 354.893,Z 480.275,A -85,B 0,C 180,E1 -13525.828,E2 -13525.828} C_VEL
LIN {X 0,Y 354.849,Z 480.248,A -85,B 0,C 180,E1 -13529.679,E2 -13529.679} C_VEL
LIN {X 0,Y 354.801,Z 480.281,A -85,B 0,C 180,E1 -13533.703,E2 -13533.703} C_VEL
LIN {X 0,Y 354.794,Z 480.291,A -85,B 0,C 180,E1 -13536.46,E2 -13536.46} C_VEL
LIN {X 0,Y 354.82,Z 480.255,A -85,B 0,C 180,E1 -13539.424,E2 -13539.424} C_VEL
LIN {X 0,Y 354.785,Z 480.286,A -85,B 0,C 180,E1 -13542.868,E2 -13542.868} C_VEL
LIN {X 0,Y 354.766,Z 480.283,A -85,B 0,C 180,E1 -13546.105,E2 -13546.105} C_VEL
LIN {X 0,Y 354.787,Z 480.284,A -85,B 0,C 180,E1 -13549.18,E2 -13549.18} C_VEL
LIN {X 0,Y 354.807,Z 480.273,A -85,B 0,C 180,E1 -13552.403,E2 -13552.403} C_VEL
LIN {X 0,Y 354.81,Z 480.229,A -85,B 0,C 180,E1 -13554.942,E2 -13554.942} C_VEL
LIN {X 0,Y 354.793,Z 480.282,A -85,B 0,C 180,E1 -13558.406,E2 -13558.406} C_VEL
LIN {X 0,Y 354.846,Z 480.26,A -85,B 0,C 180,E1 -13561.619,E2 -13561.619} C_VEL
LIN {X 0,Y 354.9,Z 480.252,A -85,B 0,C 180,E1 -13564.173,E2 -13564.173} C_VEL
LIN {X 0,Y 354.875,Z 480.417,A -85,B 0,C 180,E1 -13567.667,E2 -13567.667} C_VEL
LIN {X 0,Y 355.063,Z 481.341,A -85,B 0,C 180,E1 -13567.852,E2 -13567.852} C_VEL
LIN {X 0,Y 363.944,Z 501.901,A -85,B 0,C 180,E1 -13568.898,E2 -13568.898} C_VEL
LIN {X 0,Y 364.237,Z 505.605,A -85,B 0,C 180,E1 -13568.994,E2 -13568.994} C_VEL
LIN {X 0,Y 363.543,Z 557.178,A -85,B 0,C 180,E1 -13570.023,E2 -13570.023} C_VEL
LIN {X 0,Y 363.433,Z 570.527,A -85,B 0,C 180,E1 -13570.43,E2 -13570.43} C_VEL
LIN {X 0,Y 363.006,Z 582.676,A -85,B 0,C 180,E1 -13571.005,E2 -13571.005} C_VEL
LIN {X 0,Y 362.457,Z 595.014,A -85,B 0,C 180,E1 -13571.825,E2 -13571.825} C_VEL
LIN {X 0,Y 361.612,Z 606.509,A -85,B 0,C 180,E1 -13572.832,E2 -13572.832} C_VEL
LIN {X 0,Y 360.616,Z 617.26,A -85,B 0,C 180,E1 -13574.022,E2 -13574.022} C_VEL
LIN {X 0,Y 359.678,Z 626.462,A -85,B 0,C 180,E1 -13575.285,E2 -13575.285} C_VEL
LIN {X 0,Y 358.824,Z 634.824,A -85,B 0,C 180,E1 -13576.695,E2 -13576.695} C_VEL
LIN {X 0,Y 357.839,Z 642.942,A -85,B 0,C 180,E1 -13578.387,E2 -13578.387} C_VEL
LIN {X 0,Y 356.899,Z 650.055,A -85,B 0,C 180,E1 -13580.247,E2 -13580.247} C_VEL
LIN {X 0,Y 356.33,Z 655.431,A -85,B 0,C 180,E1 -13582.064,E2 -13582.064} C_VEL
LIN {X 0,Y 355.677,Z 659.324,A -85,B 0,C 180,E1 -13583.761,E2 -13583.761} C_VEL
LIN {X 0,Y 355.234,Z 662.191,A -85,B 0,C 180,E1 -13585.461,E2 -13585.461} C_VEL
LIN {X 0,Y 355.202,Z 663.539,A -85,B 0,C 180,E1 -13586.597,E2 -13586.597} C_VEL
LIN {X 0,Y 355.005,Z 664.522,A -85,B 0,C 180,E1 -13587.731,E2 -13587.731} C_VEL
LIN {X 0,Y 355.06,Z 665.102,A -85,B 0,C 180,E1 -13588.866,E2 -13588.866} C_VEL
LIN {X 0,Y 355.039,Z 665.33,A -85,B 0,C 180,E1 -13590,E2 -13590} C_VEL
LIN {X 0,Y 355.06,Z 665.144,A -85,B 0,C 180,E1 -13591.134,E2 -13591.134} C_VEL
LIN {X 0,Y 355.004,Z 664.591,A -85,B 0,C 180,E1 -13592.269,E2 -13592.269} C_VEL
LIN {X 0,Y 355.198,Z 663.636,A -85,B 0,C 180,E1 -13593.403,E2 -13593.403} C_VEL
LIN {X 0,Y 355.223,Z 662.332,A -85,B 0,C 180,E1 -13594.539,E2 -13594.539} C_VEL
LIN {X 0,Y 355.67,Z 659.517,A -85,B 0,C 180,E1 -13596.239,E2 -13596.239} C_VEL
LIN {X 0,Y 356.306,Z 655.691,A -85,B 0,C 180,E1 -13597.936,E2 -13597.936} C_VEL
LIN {X 0,Y 356.836,Z 650.614,A -85,B 0,C 180,E1 -13599.694,E2 -13599.694} C_VEL
LIN {X 0,Y 357.639,Z 644.586,A -85,B 0,C 180,E1 -13601.333,E2 -13601.333} C_VEL
LIN {X 0,Y 358.637,Z 636.806,A -85,B 0,C 180,E1 -13603.024,E2 -13603.024} C_VEL
LIN {X 0,Y 359.642,Z 627.136,A -85,B 0,C 180,E1 -13604.716,E2 -13604.716} C_VEL
LIN {X 0,Y 360.576,Z 618.096,A -85,B 0,C 180,E1 -13605.98,E2 -13605.98} C_VEL
LIN {X 0,Y 361.586,Z 607.594,A -85,B 0,C 180,E1 -13607.162,E2 -13607.162} C_VEL
LIN {X 0,Y 362.428,Z 595.923,A -85,B 0,C 180,E1 -13608.206,E2 -13608.206} C_VEL
LIN {X 0,Y 363.12,Z 584.475,A -85,B 0,C 180,E1 -13608.989,E2 -13608.989} C_VEL
LIN {X 0,Y 363.444,Z 572.502,A -85,B 0,C 180,E1 -13609.595,E2 -13609.595} C_VEL
LIN {X 0,Y 363.568,Z 560.767,A -85,B 0,C 180,E1 -13609.993,E2 -13609.993} C_VEL
LIN {X 0,Y 363.879,Z 524.176,A -85,B 0,C 180,E1 -13610.748,E2 -13610.748} C_VEL
LIN {X 0,Y 364.249,Z 502.663,A -85,B 0,C 180,E1 -13611.172,E2 -13611.172} C_VEL
LIN {X 0,Y 360.193,Z 492.917,A -85,B 0,C 180,E1 -13611.641,E2 -13611.641} C_VEL
LIN {X 0,Y 358.705,Z 491.097,A -85,B 0,C 180,E1 -13611.779,E2 -13611.779} C_VEL
LIN {X 0,Y 351.276,Z 487.926,A -85,B 0,C 180,E1 -13612.357,E2 -13612.357} C_VEL
LIN {X 0,Y 349.762,Z 486.121,A -85,B 0,C 180,E1 -13612.503,E2 -13612.503} C_VEL
LIN {X 0,Y 347.962,Z 481.981,A -85,B 0,C 180,E1 -13612.765,E2 -13612.765} C_VEL
LIN {X 0,Y 347.824,Z 481.194,A -85,B 0,C 180,E1 -13613.046,E2 -13613.046} C_VEL
LIN {X 0,Y 347.831,Z 481.124,A -85,B 0,C 180,E1 -13616.392,E2 -13616.392} C_VEL
LIN {X 0,Y 347.749,Z 481.169,A -85,B 0,C 180,E1 -13620.347,E2 -13620.347} C_VEL
LIN {X 0,Y 347.747,Z 481.167,A -85,B 0,C 180,E1 -13624.043,E2 -13624.043} C_VEL
LIN {X 0,Y 347.761,Z 481.152,A -85,B 0,C 180,E1 -13627.32,E2 -13627.32} C_VEL
LIN {X 0,Y 347.731,Z 481.17,A -85,B 0,C 180,E1 -13630.296,E2 -13630.296} C_VEL
LIN {X 0,Y 347.721,Z 481.153,A -85,B 0,C 180,E1 -13633.407,E2 -13633.407} C_VEL
LIN {X 0,Y 347.725,Z 481.173,A -85,B 0,C 180,E1 -13636.685,E2 -13636.685} C_VEL
LIN {X 0,Y 347.742,Z 481.133,A -85,B 0,C 180,E1 -13640.172,E2 -13640.172} C_VEL
LIN {X 0,Y 347.757,Z 481.158,A -85,B 0,C 180,E1 -13642.678,E2 -13642.678} C_VEL
LIN {X 0,Y 347.743,Z 481.161,A -85,B 0,C 180,E1 -13645.955,E2 -13645.955} C_VEL
LIN {X 0,Y 347.759,Z 481.124,A -85,B 0,C 180,E1 -13649.653,E2 -13649.653} C_VEL
LIN {X 0,Y 347.847,Z 481.145,A -85,B 0,C 180,E1 -13652.744,E2 -13652.744} C_VEL
LIN {X 0,Y 347.782,Z 481.158,A -85,B 0,C 180,E1 -13656.161,E2 -13656.161} C_VEL
LIN {X 0,Y 347.8,Z 481.16,A -85,B 0,C 180,E1 -13659.908,E2 -13659.908} C_VEL
LIN {X 0,Y 347.859,Z 481.148,A -85,B 0,C 180,E1 -13662.359,E2 -13662.359} C_VEL
LIN {X 0,Y 347.89,Z 481.148,A -85,B 0,C 180,E1 -13665.97,E2 -13665.97} C_VEL
LIN {X 0,Y 347.921,Z 481.133,A -85,B 0,C 180,E1 -13669.525,E2 -13669.525} C_VEL
LIN {X 0,Y 348.098,Z 481.12,A -85,B 0,C 180,E1 -13673.042,E2 -13673.042} C_VEL
LIN {X 0,Y 348.2,Z 481.096,A -85,B 0,C 180,E1 -13677.686,E2 -13677.686} C_VEL
LIN {X 0,Y 348.36,Z 481.088,A -85,B 0,C 180,E1 -13680,E2 -13680} C_VEL
LIN {X 0,Y 348.2,Z 481.103,A -85,B 0,C 180,E1 -13682.313,E2 -13682.313} C_VEL
LIN {X 0,Y 348.087,Z 481.122,A -85,B 0,C 180,E1 -13686.958,E2 -13686.958} C_VEL
LIN {X 0,Y 347.921,Z 481.131,A -85,B 0,C 180,E1 -13690.475,E2 -13690.475} C_VEL
LIN {X 0,Y 347.891,Z 481.149,A -85,B 0,C 180,E1 -13694.15,E2 -13694.15} C_VEL
LIN {X 0,Y 347.883,Z 481.122,A -85,B 0,C 180,E1 -13698.29,E2 -13698.29} C_VEL
LIN {X 0,Y 347.765,Z 481.164,A -85,B 0,C 180,E1 -13702.58,E2 -13702.58} C_VEL
LIN {X 0,Y 347.806,Z 481.154,A -85,B 0,C 180,E1 -13705.109,E2 -13705.109} C_VEL
LIN {X 0,Y 347.807,Z 481.142,A -85,B 0,C 180,E1 -13707.694,E2 -13707.694} C_VEL
LIN {X 0,Y 347.759,Z 481.166,A -85,B 0,C 180,E1 -13710.347,E2 -13710.347} C_VEL
LIN {X 0,Y 347.739,Z 481.165,A -85,B 0,C 180,E1 -13714.465,E2 -13714.465} C_VEL
LIN {X 0,Y 347.77,Z 481.155,A -85,B 0,C 180,E1 -13717.99,E2 -13717.99} C_VEL
LIN {X 0,Y 347.747,Z 481.158,A -85,B 0,C 180,E1 -13721.831,E2 -13721.831} C_VEL
LIN {X 0,Y 347.794,Z 481.136,A -85,B 0,C 180,E1 -13725.012,E2 -13725.012} C_VEL
LIN {X 0,Y 347.781,Z 481.153,A -85,B 0,C 180,E1 -13728.392,E2 -13728.392} C_VEL
LIN {X 0,Y 347.774,Z 481.165,A -85,B 0,C 180,E1 -13732.012,E2 -13732.012} C_VEL
LIN {X 0,Y 347.792,Z 481.361,A -85,B 0,C 180,E1 -13733.895,E2 -13733.895} C_VEL
LIN {X 0,Y 350.757,Z 493.124,A -85,B 0,C 180,E1 -13736.565,E2 -13736.565} C_VEL
LIN {X 0,Y 353.918,Z 507.328,A -85,B 0,C 180,E1 -13739.578,E2 -13739.578} C_VEL
LIN {X 0,Y 354.162,Z 510.788,A -85,B 0,C 180,E1 -13740.258,E2 -13740.258} C_VEL
LIN {X 0,Y 351.98,Z 530.971,A -85,B 0,C 180,E1 -13743.964,E2 -13743.964} C_VEL
LIN {X 0,Y 350.49,Z 546.914,A -85,B 0,C 180,E1 -13746.89,E2 -13746.89} C_VEL
LIN {X 0,Y 351.251,Z 553.536,A -85,B 0,C 180,E1 -13747.133,E2 -13747.133} C_VEL
LIN {X 0,Y 355.117,Z 587.107,A -85,B 0,C 180,E1 -13748.097,E2 -13748.097} C_VEL
LIN {X 0,Y 356.176,Z 600.838,A -85,B 0,C 180,E1 -13748.452,E2 -13748.452} C_VEL
LIN {X 0,Y 355.11,Z 658.033,A -85,B 0,C 180,E1 -13749.623,E2 -13749.623} C_VEL
LIN {X 0,Y 354.486,Z 671.312,A -85,B 0,C 180,E1 -13750.115,E2 -13750.115} C_VEL
LIN {X 0,Y 353.41,Z 683.492,A -85,B 0,C 180,E1 -13750.77,E2 -13750.77} C_VEL
LIN {X 0,Y 352.159,Z 695.827,A -85,B 0,C 180,E1 -13751.681,E2 -13751.681} C_VEL
LIN {X 0,Y 350.891,Z 707.531,A -85,B 0,C 180,E1 -13752.817,E2 -13752.817} C_VEL
LIN {X 0,Y 349.643,Z 718.096,A -85,B 0,C 180,E1 -13754.106,E2 -13754.106} C_VEL
LIN {X 0,Y 348.589,Z 726.788,A -85,B 0,C 180,E1 -13755.408,E2 -13755.408} C_VEL
LIN {X 0,Y 347.875,Z 734.819,A -85,B 0,C 180,E1 -13756.863,E2 -13756.863} C_VEL
LIN {X 0,Y 347.199,Z 742.714,A -85,B 0,C 180,E1 -13758.618,E2 -13758.618} C_VEL
LIN {X 0,Y 346.835,Z 750.043,A -85,B 0,C 180,E1 -13760.671,E2 -13760.671} C_VEL
LIN {X 0,Y 346.795,Z 754.956,A -85,B 0,C 180,E1 -13762.431,E2 -13762.431} C_VEL
LIN {X 0,Y 346.887,Z 758.731,A -85,B 0,C 180,E1 -13764.186,E2 -13764.186} C_VEL
LIN {X 0,Y 347.057,Z 760.696,A -85,B 0,C 180,E1 -13765.354,E2 -13765.354} C_VEL
LIN {X 0,Y 347.172,Z 762.168,A -85,B 0,C 180,E1 -13766.518,E2 -13766.518} C_VEL
LIN {X 0,Y 347.603,Z 763.901,A -85,B 0,C 180,E1 -13768.842,E2 -13768.842} C_VEL
LIN {X 0,Y 347.683,Z 764.136,A -85,B 0,C 180,E1 -13770,E2 -13770} C_VEL
LIN {X 0,Y 347.603,Z 763.897,A -85,B 0,C 180,E1 -13771.158,E2 -13771.158} C_VEL
LIN {X 0,Y 347.176,Z 762.161,A -85,B 0,C 180,E1 -13773.482,E2 -13773.482} C_VEL
LIN {X 0,Y 347.063,Z 760.685,A -85,B 0,C 180,E1 -13774.646,E2 -13774.646} C_VEL
LIN {X 0,Y 346.824,Z 756.678,A -85,B 0,C 180,E1 -13776.815,E2 -13776.815} C_VEL
LIN {X 0,Y 346.799,Z 751.772,A -85,B 0,C 180,E1 -13778.742,E2 -13778.742} C_VEL
LIN {X 0,Y 346.944,Z 746.031,A -85,B 0,C 180,E1 -13780.504,E2 -13780.504} C_VEL
LIN {X 0,Y 347.497,Z 738.931,A -85,B 0,C 180,E1 -13782.26,E2 -13782.26} C_VEL
LIN {X 0,Y 348.375,Z 730.091,A -85,B 0,C 180,E1 -13784.009,E2 -13784.009} C_VEL
LIN {X 0,Y 349.338,Z 721.067,A -85,B 0,C 180,E1 -13785.46,E2 -13785.46} C_VEL
LIN {X 0,Y 350.217,Z 712.379,A -85,B 0,C 180,E1 -13786.616,E2 -13786.616} C_VEL
LIN {X 0,Y 351.702,Z 700.453,A -85,B 0,C 180,E1 -13787.892,E2 -13787.892} C_VEL
LIN {X 0,Y 352.983,Z 688.466,A -85,B 0,C 180,E1 -13788.877,E2 -13788.877} C_VEL
LIN {X 0,Y 354.08,Z 676.022,A -85,B 0,C 180,E1 -13789.644,E2 -13789.644} C_VEL
LIN {X 0,Y 354.888,Z 663.24,A -85,B 0,C 180,E1 -13790.201,E2 -13790.201} C_VEL
LIN {X 0,Y 355.27,Z 649.8,A -85,B 0,C 180,E1 -13790.556,E2 -13790.556} C_VEL
LIN {X 0,Y 356.092,Z 598.301,A -85,B 0,C 180,E1 -13791.592,E2 -13791.592} C_VEL
LIN {X 0,Y 352.354,Z 562.51,A -85,B 0,C 180,E1 -13792.587,E2 -13792.587} C_VEL
LIN {X 0,Y 350.477,Z 547.127,A -85,B 0,C 180,E1 -13793.071,E2 -13793.071} C_VEL
LIN {X 0,Y 352.496,Z 525.768,A -85,B 0,C 180,E1 -13796.973,E2 -13796.973} C_VEL
LIN {X 0,Y 354.165,Z 510.702,A -85,B 0,C 180,E1 -13799.741,E2 -13799.741} C_VEL
LIN {X 0,Y 353.882,Z 507.232,A -85,B 0,C 180,E1 -13800.425,E2 -13800.425} C_VEL
LIN {X 0,Y 350.731,Z 493.014,A -85,B 0,C 180,E1 -13803.437,E2 -13803.437} C_VEL
LIN {X 0,Y 347.791,Z 481.316,A -85,B 0,C 180,E1 -13806.094,E2 -13806.094} C_VEL
LIN {X 0,Y 347.783,Z 481.144,A -85,B 0,C 180,E1 -13809.834,E2 -13809.834} C_VEL
LIN {X 0,Y 347.783,Z 481.165,A -85,B 0,C 180,E1 -13813.397,E2 -13813.397} C_VEL
LIN {X 0,Y 347.725,Z 481.141,A -85,B 0,C 180,E1 -13816.685,E2 -13816.685} C_VEL
LIN {X 0,Y 347.743,Z 481.168,A -85,B 0,C 180,E1 -13820.172,E2 -13820.172} C_VEL
LIN {X 0,Y 347.758,Z 481.161,A -85,B 0,C 180,E1 -13822.679,E2 -13822.679} C_VEL
LIN {X 0,Y 347.743,Z 481.158,A -85,B 0,C 180,E1 -13825.956,E2 -13825.956} C_VEL
LIN {X 0,Y 347.759,Z 481.166,A -85,B 0,C 180,E1 -13829.653,E2 -13829.653} C_VEL
LIN {X 0,Y 347.846,Z 481.134,A -85,B 0,C 180,E1 -13832.744,E2 -13832.744} C_VEL
LIN {X 0,Y 347.782,Z 481.162,A -85,B 0,C 180,E1 -13836.161,E2 -13836.161} C_VEL
LIN {X 0,Y 347.793,Z 481.14,A -85,B 0,C 180,E1 -13839.908,E2 -13839.908} C_VEL
LIN {X 0,Y 347.859,Z 481.131,A -85,B 0,C 180,E1 -13842.359,E2 -13842.359} C_VEL
LIN {X 0,Y 347.89,Z 481.15,A -85,B 0,C 180,E1 -13845.971,E2 -13845.971} C_VEL
LIN {X 0,Y 347.921,Z 481.133,A -85,B 0,C 180,E1 -13849.525,E2 -13849.525} C_VEL
LIN {X 0,Y 348.087,Z 481.123,A -85,B 0,C 180,E1 -13853.042,E2 -13853.042} C_VEL
LIN {X 0,Y 348.2,Z 481.106,A -85,B 0,C 180,E1 -13857.687,E2 -13857.687} C_VEL
LIN {X 0,Y 348.361,Z 481.09,A -85,B 0,C 180,E1 -13860,E2 -13860} C_VEL
LIN {X 0,Y 348.201,Z 481.097,A -85,B 0,C 180,E1 -13862.314,E2 -13862.314} C_VEL
LIN {X 0,Y 348.087,Z 481.122,A -85,B 0,C 180,E1 -13866.958,E2 -13866.958} C_VEL
LIN {X 0,Y 347.921,Z 481.133,A -85,B 0,C 180,E1 -13870.475,E2 -13870.475} C_VEL
LIN {X 0,Y 347.891,Z 481.148,A -85,B 0,C 180,E1 -13874.15,E2 -13874.15} C_VEL
LIN {X 0,Y 347.884,Z 481.147,A -85,B 0,C 180,E1 -13878.29,E2 -13878.29} C_VEL
LIN {X 0,Y 347.771,Z 481.154,A -85,B 0,C 180,E1 -13881.631,E2 -13881.631} C_VEL
LIN {X 0,Y 347.806,Z 481.161,A -85,B 0,C 180,E1 -13885.109,E2 -13885.109} C_VEL
LIN {X 0,Y 347.806,Z 481.149,A -85,B 0,C 180,E1 -13887.694,E2 -13887.694} C_VEL
LIN {X 0,Y 347.759,Z 481.124,A -85,B 0,C 180,E1 -13890.347,E2 -13890.347} C_VEL
LIN {X 0,Y 347.74,Z 481.163,A -85,B 0,C 180,E1 -13894.465,E2 -13894.465} C_VEL
LIN {X 0,Y 347.769,Z 481.155,A -85,B 0,C 180,E1 -13897.989,E2 -13897.989} C_VEL
LIN {X 0,Y 347.747,Z 481.154,A -85,B 0,C 180,E1 -13901.831,E2 -13901.831} C_VEL
LIN {X 0,Y 347.763,Z 481.162,A -85,B 0,C 180,E1 -13905.018,E2 -13905.018} C_VEL
LIN {X 0,Y 347.748,Z 481.152,A -85,B 0,C 180,E1 -13908.398,E2 -13908.398} C_VEL
LIN {X 0,Y 347.773,Z 481.158,A -85,B 0,C 180,E1 -13912.012,E2 -13912.012} C_VEL
LIN {X 0,Y 347.743,Z 481.106,A -85,B 0,C 180,E1 -13915.537,E2 -13915.537} C_VEL
LIN {X 0,Y 347.76,Z 481.17,A -85,B 0,C 180,E1 -13919.654,E2 -13919.654} C_VEL
LIN {X 0,Y 347.831,Z 481.124,A -85,B 0,C 180,E1 -13923.608,E2 -13923.608} C_VEL
LIN {X 0,Y 347.838,Z 481.296,A -85,B 0,C 180,E1 -13927.19,E2 -13927.19} C_VEL
LIN {X 0,Y 348.019,Z 482.209,A -85,B 0,C 180,E1 -13927.374,E2 -13927.374} C_VEL
LIN {X 0,Y 357.547,Z 504.118,A -85,B 0,C 180,E1 -13928.528,E2 -13928.528} C_VEL
LIN {X 0,Y 356.885,Z 562.847,A -85,B 0,C 180,E1 -13929.751,E2 -13929.751} C_VEL
LIN {X 0,Y 356.708,Z 575.622,A -85,B 0,C 180,E1 -13930.225,E2 -13930.225} C_VEL
LIN {X 0,Y 356.213,Z 588.34,A -85,B 0,C 180,E1 -13930.928,E2 -13930.928} C_VEL
LIN {X 0,Y 355.504,Z 600.663,A -85,B 0,C 180,E1 -13931.857,E2 -13931.857} C_VEL
LIN {X 0,Y 354.427,Z 612.234,A -85,B 0,C 180,E1 -13932.994,E2 -13932.994} C_VEL
LIN {X 0,Y 353.411,Z 622.561,A -85,B 0,C 180,E1 -13934.28,E2 -13934.28} C_VEL
LIN {X 0,Y 352.489,Z 630.985,A -85,B 0,C 180,E1 -13935.569,E2 -13935.569} C_VEL
LIN {X 0,Y 351.635,Z 638.722,A -85,B 0,C 180,E1 -13937.006,E2 -13937.006} C_VEL
LIN {X 0,Y 350.612,Z 646.401,A -85,B 0,C 180,E1 -13938.759,E2 -13938.759} C_VEL
LIN {X 0,Y 349.863,Z 652.152,A -85,B 0,C 180,E1 -13940.401,E2 -13940.401} C_VEL
LIN {X 0,Y 349.371,Z 656.42,A -85,B 0,C 180,E1 -13941.905,E2 -13941.905} C_VEL
LIN {X 0,Y 348.691,Z 660.313,A -85,B 0,C 180,E1 -13943.636,E2 -13943.636} C_VEL
LIN {X 0,Y 348.225,Z 663.18,A -85,B 0,C 180,E1 -13945.37,E2 -13945.37} C_VEL
LIN {X 0,Y 348.186,Z 664.528,A -85,B 0,C 180,E1 -13946.528,E2 -13946.528} C_VEL
LIN {X 0,Y 348.035,Z 666.09,A -85,B 0,C 180,E1 -13948.843,E2 -13948.843} C_VEL
LIN {X 0,Y 348.013,Z 666.317,A -85,B 0,C 180,E1 -13950,E2 -13950} C_VEL
LIN {X 0,Y 348.035,Z 666.132,A -85,B 0,C 180,E1 -13951.157,E2 -13951.157} C_VEL
LIN {X 0,Y 347.983,Z 665.578,A -85,B 0,C 180,E1 -13952.315,E2 -13952.315} C_VEL
LIN {X 0,Y 348.182,Z 664.624,A -85,B 0,C 180,E1 -13953.472,E2 -13953.472} C_VEL
LIN {X 0,Y 348.215,Z 663.32,A -85,B 0,C 180,E1 -13954.631,E2 -13954.631} C_VEL
LIN {X 0,Y 348.684,Z 660.504,A -85,B 0,C 180,E1 -13956.365,E2 -13956.365} C_VEL
LIN {X 0,Y 349.346,Z 656.678,A -85,B 0,C 180,E1 -13958.095,E2 -13958.095} C_VEL
LIN {X 0,Y 349.91,Z 651.601,A -85,B 0,C 180,E1 -13959.888,E2 -13959.888} C_VEL
LIN {X 0,Y 350.75,Z 645.572,A -85,B 0,C 180,E1 -13961.558,E2 -13961.558} C_VEL
LIN {X 0,Y 351.793,Z 637.792,A -85,B 0,C 180,E1 -13963.282,E2 -13963.282} C_VEL
LIN {X 0,Y 352.847,Z 628.121,A -85,B 0,C 180,E1 -13965.006,E2 -13965.006} C_VEL
LIN {X 0,Y 353.823,Z 619.081,A -85,B 0,C 180,E1 -13966.294,E2 -13966.294} C_VEL
LIN {X 0,Y 354.877,Z 608.577,A -85,B 0,C 180,E1 -13967.496,E2 -13967.496} C_VEL
LIN {X 0,Y 355.736,Z 597.062,A -85,B 0,C 180,E1 -13968.547,E2 -13968.547} C_VEL
LIN {X 0,Y 356.47,Z 585.791,A -85,B 0,C 180,E1 -13969.335,E2 -13969.335} C_VEL
LIN {X 0,Y 356.815,Z 573.479,A -85,B 0,C 180,E1 -13969.975,E2 -13969.975} C_VEL
LIN {X 0,Y 356.945,Z 561.738,A -85,B 0,C 180,E1 -13970.38,E2 -13970.38} C_VEL
LIN {X 0,Y 357.337,Z 522.469,A -85,B 0,C 180,E1 -13971.202,E2 -13971.202} C_VEL
LIN {X 0,Y 357.573,Z 504.178,A -85,B 0,C 180,E1 -13971.576,E2 -13971.576} C_VEL
LIN {X 0,Y 349.762,Z 486.121,A -85,B 0,C 180,E1 -13972.503,E2 -13972.503} C_VEL
LIN {X 0,Y 348.467,Z 483.885,A -85,B 0,C 180,E1 -13972.759,E2 -13972.759} C_VEL
LIN {X 0,Y 346.656,Z 482.29,A -85,B 0,C 180,E1 -13973.285,E2 -13973.285} C_VEL
LIN {X 0,Y 344.41,Z 481.653,A -85,B 0,C 180,E1 -13974.164,E2 -13974.164} C_VEL
LIN {X 0,Y 341.634,Z 481.901,A -85,B 0,C 180,E1 -13975.927,E2 -13975.927} C_VEL
LIN {X 0,Y 340.779,Z 481.997,A -85,B 0,C 180,E1 -13977.425,E2 -13977.425} C_VEL
LIN {X 0,Y 340.697,Z 482.044,A -85,B 0,C 180,E1 -13981.044,E2 -13981.044} C_VEL
LIN {X 0,Y 340.717,Z 482.04,A -85,B 0,C 180,E1 -13985.278,E2 -13985.278} C_VEL
LIN {X 0,Y 340.708,Z 482.039,A -85,B 0,C 180,E1 -13988.385,E2 -13988.385} C_VEL
LIN {X 0,Y 340.696,Z 482.027,A -85,B 0,C 180,E1 -13992.045,E2 -13992.045} C_VEL
LIN {X 0,Y 340.682,Z 482.051,A -85,B 0,C 180,E1 -13995.461,E2 -13995.461} C_VEL
LIN {X 0,Y 340.681,Z 482.025,A -85,B 0,C 180,E1 -13998.689,E2 -13998.689} C_VEL
LIN {X 0,Y 340.728,Z 482.024,A -85,B 0,C 180,E1 -14001.772,E2 -14001.772} C_VEL
LIN {X 0,Y 340.718,Z 482.038,A -85,B 0,C 180,E1 -14005.595,E2 -14005.595} C_VEL
LIN {X 0,Y 340.698,Z 482.002,A -85,B 0,C 180,E1 -14008.955,E2 -14008.955} C_VEL
LIN {X 0,Y 340.774,Z 482.025,A -85,B 0,C 180,E1 -14012.473,E2 -14012.473} C_VEL
LIN {X 0,Y 340.75,Z 482.036,A -85,B 0,C 180,E1 -14015.638,E2 -14015.638} C_VEL
LIN {X 0,Y 340.73,Z 482.04,A -85,B 0,C 180,E1 -14019.473,E2 -14019.473} C_VEL
LIN {X 0,Y 340.85,Z 482.021,A -85,B 0,C 180,E1 -14021.984,E2 -14021.984} C_VEL
LIN {X 0,Y 340.862,Z 482.024,A -85,B 0,C 180,E1 -14025.705,E2 -14025.705} C_VEL
LIN {X 0,Y 340.863,Z 482.015,A -85,B 0,C 180,E1 -14029.306,E2 -14029.306} C_VEL
LIN {X 0,Y 341.067,Z 481.994,A -85,B 0,C 180,E1 -14032.898,E2 -14032.898} C_VEL
LIN {X 0,Y 341.162,Z 481.971,A -85,B 0,C 180,E1 -14037.639,E2 -14037.639} C_VEL
LIN {X 0,Y 341.309,Z 481.966,A -85,B 0,C 180,E1 -14040,E2 -14040} C_VEL
LIN {X 0,Y 341.162,Z 481.979,A -85,B 0,C 180,E1 -14042.361,E2 -14042.361} C_VEL
LIN {X 0,Y 341.055,Z 481.999,A -85,B 0,C 180,E1 -14047.102,E2 -14047.102} C_VEL
LIN {X 0,Y 340.863,Z 482.01,A -85,B 0,C 180,E1 -14050.694,E2 -14050.694} C_VEL
LIN {X 0,Y 340.856,Z 482.025,A -85,B 0,C 180,E1 -14054.325,E2 -14054.325} C_VEL
LIN {X 0,Y 340.829,Z 481.999,A -85,B 0,C 180,E1 -14058.466,E2 -14058.466} C_VEL
LIN {X 0,Y 340.717,Z 482.041,A -85,B 0,C 180,E1 -14061.845,E2 -14061.845} C_VEL
LIN {X 0,Y 340.766,Z 482.021,A -85,B 0,C 180,E1 -14065.665,E2 -14065.665} C_VEL
LIN {X 0,Y 340.737,Z 482.032,A -85,B 0,C 180,E1 -14068.32,E2 -14068.32} C_VEL
LIN {X 0,Y 340.699,Z 482.045,A -85,B 0,C 180,E1 -14071.045,E2 -14071.045} C_VEL
LIN {X 0,Y 340.713,Z 482.042,A -85,B 0,C 180,E1 -14075.28,E2 -14075.28} C_VEL
LIN {X 0,Y 340.705,Z 482.035,A -85,B 0,C 180,E1 -14078.387,E2 -14078.387} C_VEL
LIN {X 0,Y 340.695,Z 482.034,A -85,B 0,C 180,E1 -14082.046,E2 -14082.046} C_VEL
LIN {X 0,Y 340.718,Z 482.024,A -85,B 0,C 180,E1 -14085.469,E2 -14085.469} C_VEL
LIN {X 0,Y 340.722,Z 482.027,A -85,B 0,C 180,E1 -14088.697,E2 -14088.697} C_VEL
LIN {X 0,Y 340.737,Z 482.045,A -85,B 0,C 180,E1 -14091.774,E2 -14091.774} C_VEL
LIN {X 0,Y 340.758,Z 482.286,A -85,B 0,C 180,E1 -14093.45,E2 -14093.45} C_VEL
LIN {X 0,Y 343.702,Z 493.832,A -85,B 0,C 180,E1 -14096.14,E2 -14096.14} C_VEL
LIN {X 0,Y 346.898,Z 508.292,A -85,B 0,C 180,E1 -14099.287,E2 -14099.287} C_VEL
LIN {X 0,Y 347.305,Z 511.262,A -85,B 0,C 180,E1 -14099.898,E2 -14099.898} C_VEL
LIN {X 0,Y 345.427,Z 528.208,A -85,B 0,C 180,E1 -14103.084,E2 -14103.084} C_VEL
LIN {X 0,Y 343.684,Z 546.189,A -85,B 0,C 180,E1 -14106.436,E2 -14106.436} C_VEL
LIN {X 0,Y 347.742,Z 580.614,A -85,B 0,C 180,E1 -14107.49,E2 -14107.49} C_VEL
LIN {X 0,Y 349.539,Z 601.439,A -85,B 0,C 180,E1 -14108.056,E2 -14108.056} C_VEL
LIN {X 0,Y 348.455,Z 657.047,A -85,B 0,C 180,E1 -14109.216,E2 -14109.216} C_VEL
LIN {X 0,Y 347.819,Z 670.322,A -85,B 0,C 180,E1 -14109.717,E2 -14109.717} C_VEL
LIN {X 0,Y 346.69,Z 682.496,A -85,B 0,C 180,E1 -14110.382,E2 -14110.382} C_VEL
LIN {X 0,Y 345.423,Z 694.833,A -85,B 0,C 180,E1 -14111.31,E2 -14111.31} C_VEL
LIN {X 0,Y 344.161,Z 705.213,A -85,B 0,C 180,E1 -14112.317,E2 -14112.317} C_VEL
LIN {X 0,Y 342.962,Z 714.912,A -85,B 0,C 180,E1 -14113.482,E2 -14113.482} C_VEL
LIN {X 0,Y 341.887,Z 724.477,A -85,B 0,C 180,E1 -14114.894,E2 -14114.894} C_VEL
LIN {X 0,Y 341.254,Z 730.775,A -85,B 0,C 180,E1 -14115.997,E2 -14115.997} C_VEL
LIN {X 0,Y 340.373,Z 739.243,A -85,B 0,C 180,E1 -14117.782,E2 -14117.782} C_VEL
LIN {X 0,Y 339.863,Z 746.113,A -85,B 0,C 180,E1 -14119.576,E2 -14119.576} C_VEL
LIN {X 0,Y 339.712,Z 752.459,A -85,B 0,C 180,E1 -14121.674,E2 -14121.674} C_VEL
LIN {X 0,Y 339.747,Z 756.006,A -85,B 0,C 180,E1 -14123.182,E2 -14123.182} C_VEL
LIN {X 0,Y 339.997,Z 759.7,A -85,B 0,C 180,E1 -14125.257,E2 -14125.257} C_VEL
LIN {X 0,Y 340.124,Z 761.176,A -85,B 0,C 180,E1 -14126.446,E2 -14126.446} C_VEL
LIN {X 0,Y 340.568,Z 762.912,A -85,B 0,C 180,E1 -14128.818,E2 -14128.818} C_VEL
LIN {X 0,Y 340.657,Z 763.148,A -85,B 0,C 180,E1 -14130,E2 -14130} C_VEL
LIN {X 0,Y 340.569,Z 762.908,A -85,B 0,C 180,E1 -14131.182,E2 -14131.182} C_VEL
LIN {X 0,Y 340.127,Z 761.168,A -85,B 0,C 180,E1 -14133.554,E2 -14133.554} C_VEL
LIN {X 0,Y 340.002,Z 759.688,A -85,B 0,C 180,E1 -14134.743,E2 -14134.743} C_VEL
LIN {X 0,Y 339.766,Z 755.926,A -85,B 0,C 180,E1 -14136.844,E2 -14136.844} C_VEL
LIN {X 0,Y 339.725,Z 750.764,A -85,B 0,C 180,E1 -14138.926,E2 -14138.926} C_VEL
LIN {X 0,Y 339.891,Z 745.021,A -85,B 0,C 180,E1 -14140.725,E2 -14140.725} C_VEL
LIN {X 0,Y 340.488,Z 737.92,A -85,B 0,C 180,E1 -14142.517,E2 -14142.517} C_VEL
LIN {X 0,Y 341.27,Z 730.711,A -85,B 0,C 180,E1 -14144.003,E2 -14144.003} C_VEL
LIN {X 0,Y 342.199,Z 722.039,A -85,B 0,C 180,E1 -14145.485,E2 -14145.485} C_VEL
LIN {X 0,Y 343.23,Z 712.561,A -85,B 0,C 180,E1 -14146.811,E2 -14146.811} C_VEL
LIN {X 0,Y 344.755,Z 700.889,A -85,B 0,C 180,E1 -14148.112,E2 -14148.112} C_VEL
LIN {X 0,Y 346.048,Z 689.409,A -85,B 0,C 180,E1 -14149.116,E2 -14149.116} C_VEL
LIN {X 0,Y 347.179,Z 677.628,A -85,B 0,C 180,E1 -14149.897,E2 -14149.897} C_VEL
LIN {X 0,Y 348.134,Z 664.075,A -85,B 0,C 180,E1 -14150.533,E2 -14150.533} C_VEL
LIN {X 0,Y 348.581,Z 650.574,A -85,B 0,C 180,E1 -14150.93,E2 -14150.93} C_VEL
LIN {X 0,Y 349.47,Z 598.971,A -85,B 0,C 180,E1 -14151.986,E2 -14151.986} C_VEL
LIN {X 0,Y 345.67,Z 562.483,A -85,B 0,C 180,E1 -14153.026,E2 -14153.026} C_VEL
LIN {X 0,Y 343.666,Z 546.084,A -85,B 0,C 180,E1 -14153.557,E2 -14153.557} C_VEL
LIN {X 0,Y 346.002,Z 523.112,A -85,B 0,C 180,E1 -14157.85,E2 -14157.85} C_VEL
LIN {X 0,Y 347.292,Z 511.188,A -85,B 0,C 180,E1 -14160.099,E2 -14160.099} C_VEL
LIN {X 0,Y 345.333,Z 500.907,A -85,B 0,C 180,E1 -14162.274,E2 -14162.274} C_VEL
LIN {X 0,Y 342.022,Z 487.08,A -85,B 0,C 180,E1 -14165.382,E2 -14165.382} C_VEL
LIN {X 0,Y 340.746,Z 482.146,A -85,B 0,C 180,E1 -14166.588,E2 -14166.588} C_VEL
LIN {X 0,Y 340.761,Z 482.017,A -85,B 0,C 180,E1 -14170.261,E2 -14170.261} C_VEL
LIN {X 0,Y 340.716,Z 482.038,A -85,B 0,C 180,E1 -14173.784,E2 -14173.784} C_VEL
LIN {X 0,Y 340.674,Z 482.023,A -85,B 0,C 180,E1 -14177.095,E2 -14177.095} C_VEL
LIN {X 0,Y 340.695,Z 482.044,A -85,B 0,C 180,E1 -14180.247,E2 -14180.247} C_VEL
LIN {X 0,Y 340.705,Z 482.043,A -85,B 0,C 180,E1 -14183.559,E2 -14183.559} C_VEL
LIN {X 0,Y 340.687,Z 482.035,A -85,B 0,C 180,E1 -14186.153,E2 -14186.153} C_VEL
LIN {X 0,Y 340.77,Z 482.037,A -85,B 0,C 180,E1 -14190.332,E2 -14190.332} C_VEL
LIN {X 0,Y 340.799,Z 482.01,A -85,B 0,C 180,E1 -14193.019,E2 -14193.019} C_VEL
LIN {X 0,Y 340.749,Z 482.035,A -85,B 0,C 180,E1 -14195.638,E2 -14195.638} C_VEL
LIN {X 0,Y 340.726,Z 482.027,A -85,B 0,C 180,E1 -14199.473,E2 -14199.473} C_VEL
LIN {X 0,Y 340.85,Z 482,A -85,B 0,C 180,E1 -14201.984,E2 -14201.984} C_VEL
LIN {X 0,Y 340.862,Z 482.024,A -85,B 0,C 180,E1 -14205.705,E2 -14205.705} C_VEL
LIN {X 0,Y 340.863,Z 482.012,A -85,B 0,C 180,E1 -14209.306,E2 -14209.306} C_VEL
LIN {X 0,Y 341.055,Z 482,A -85,B 0,C 180,E1 -14212.898,E2 -14212.898} C_VEL
LIN {X 0,Y 341.162,Z 481.982,A -85,B 0,C 180,E1 -14217.639,E2 -14217.639} C_VEL
LIN {X 0,Y 341.309,Z 481.968,A -85,B 0,C 180,E1 -14220,E2 -14220} C_VEL
LIN {X 0,Y 341.163,Z 481.973,A -85,B 0,C 180,E1 -14222.361,E2 -14222.361} C_VEL
LIN {X 0,Y 341.055,Z 481.997,A -85,B 0,C 180,E1 -14227.102,E2 -14227.102} C_VEL
LIN {X 0,Y 340.863,Z 482.014,A -85,B 0,C 180,E1 -14230.694,E2 -14230.694} C_VEL
LIN {X 0,Y 340.856,Z 482.024,A -85,B 0,C 180,E1 -14234.325,E2 -14234.325} C_VEL
LIN {X 0,Y 340.83,Z 482.027,A -85,B 0,C 180,E1 -14238.467,E2 -14238.467} C_VEL
LIN {X 0,Y 340.717,Z 482.032,A -85,B 0,C 180,E1 -14241.845,E2 -14241.845} C_VEL
LIN {X 0,Y 340.767,Z 482.035,A -85,B 0,C 180,E1 -14245.665,E2 -14245.665} C_VEL
LIN {X 0,Y 340.736,Z 482.021,A -85,B 0,C 180,E1 -14248.32,E2 -14248.32} C_VEL
LIN {X 0,Y 340.698,Z 482.001,A -85,B 0,C 180,E1 -14251.045,E2 -14251.045} C_VEL
LIN {X 0,Y 340.713,Z 482.045,A -85,B 0,C 180,E1 -14255.28,E2 -14255.28} C_VEL
LIN {X 0,Y 340.705,Z 482.025,A -85,B 0,C 180,E1 -14258.387,E2 -14258.387} C_VEL
LIN {X 0,Y 340.695,Z 482.036,A -85,B 0,C 180,E1 -14262.046,E2 -14262.046} C_VEL
LIN {X 0,Y 340.68,Z 482.04,A -85,B 0,C 180,E1 -14265.462,E2 -14265.462} C_VEL
LIN {X 0,Y 340.684,Z 482.033,A -85,B 0,C 180,E1 -14268.691,E2 -14268.691} C_VEL
LIN {X 0,Y 340.732,Z 482.035,A -85,B 0,C 180,E1 -14271.774,E2 -14271.774} C_VEL
LIN {X 0,Y 340.722,Z 481.979,A -85,B 0,C 180,E1 -14275.596,E2 -14275.596} C_VEL
LIN {X 0,Y 340.768,Z 482.04,A -85,B 0,C 180,E1 -14280.021,E2 -14280.021} C_VEL
LIN {X 0,Y 340.803,Z 481.995,A -85,B 0,C 180,E1 -14283.021,E2 -14283.021} C_VEL
LIN {X 0,Y 340.78,Z 482.18,A -85,B 0,C 180,E1 -14286.69,E2 -14286.69} C_VEL
LIN {X 0,Y 341.013,Z 483.176,A -85,B 0,C 180,E1 -14286.883,E2 -14286.883} C_VEL
LIN {X 0,Y 350.95,Z 505.821,A -85,B 0,C 180,E1 -14288.119,E2 -14288.119} C_VEL
LIN {X 0,Y 350.281,Z 562.975,A -85,B 0,C 180,E1 -14289.329,E2 -14289.329} C_VEL
LIN {X 0,Y 350.104,Z 576.012,A -85,B 0,C 180,E1 -14289.804,E2 -14289.804} C_VEL
LIN {X 0,Y 349.629,Z 588.22,A -85,B 0,C 180,E1 -14290.478,E2 -14290.478} C_VEL
LIN {X 0,Y 348.895,Z 600.564,A -85,B 0,C 180,E1 -14291.404,E2 -14291.404} C_VEL
LIN {X 0,Y 347.943,Z 610.619,A -85,B 0,C 180,E1 -14292.364,E2 -14292.364} C_VEL
LIN {X 0,Y 346.848,Z 621.459,A -85,B 0,C 180,E1 -14293.672,E2 -14293.672} C_VEL
LIN {X 0,Y 345.686,Z 631.976,A -85,B 0,C 180,E1 -14295.278,E2 -14295.278} C_VEL
LIN {X 0,Y 344.79,Z 639.713,A -85,B 0,C 180,E1 -14296.744,E2 -14296.744} C_VEL
LIN {X 0,Y 343.721,Z 647.391,A -85,B 0,C 180,E1 -14298.531,E2 -14298.531} C_VEL
LIN {X 0,Y 342.936,Z 653.142,A -85,B 0,C 180,E1 -14300.205,E2 -14300.205} C_VEL
LIN {X 0,Y 342.415,Z 657.41,A -85,B 0,C 180,E1 -14301.74,E2 -14301.74} C_VEL
LIN {X 0,Y 341.707,Z 661.302,A -85,B 0,C 180,E1 -14303.505,E2 -14303.505} C_VEL
LIN {X 0,Y 341.218,Z 664.17,A -85,B 0,C 180,E1 -14305.274,E2 -14305.274} C_VEL
LIN {X 0,Y 341.17,Z 665.517,A -85,B 0,C 180,E1 -14306.457,E2 -14306.457} C_VEL
LIN {X 0,Y 341.01,Z 667.078,A -85,B 0,C 180,E1 -14308.819,E2 -14308.819} C_VEL
LIN {X 0,Y 340.987,Z 667.305,A -85,B 0,C 180,E1 -14310,E2 -14310} C_VEL
LIN {X 0,Y 341.009,Z 667.12,A -85,B 0,C 180,E1 -14311.181,E2 -14311.181} C_VEL
LIN {X 0,Y 341.166,Z 665.612,A -85,B 0,C 180,E1 -14313.543,E2 -14313.543} C_VEL
LIN {X 0,Y 341.207,Z 664.308,A -85,B 0,C 180,E1 -14314.726,E2 -14314.726} C_VEL
LIN {X 0,Y 341.7,Z 661.491,A -85,B 0,C 180,E1 -14316.495,E2 -14316.495} C_VEL
LIN {X 0,Y 342.39,Z 657.665,A -85,B 0,C 180,E1 -14318.261,E2 -14318.261} C_VEL
LIN {X 0,Y 342.989,Z 652.587,A -85,B 0,C 180,E1 -14320.089,E2 -14320.089} C_VEL
LIN {X 0,Y 343.868,Z 646.558,A -85,B 0,C 180,E1 -14321.793,E2 -14321.793} C_VEL
LIN {X 0,Y 344.956,Z 638.777,A -85,B 0,C 180,E1 -14323.55,E2 -14323.55} C_VEL
LIN {X 0,Y 346.062,Z 629.106,A -85,B 0,C 180,E1 -14325.308,E2 -14325.308} C_VEL
LIN {X 0,Y 347.081,Z 620.065,A -85,B 0,C 180,E1 -14326.619,E2 -14326.619} C_VEL
LIN {X 0,Y 348.172,Z 609.563,A -85,B 0,C 180,E1 -14327.844,E2 -14327.844} C_VEL
LIN {X 0,Y 349.104,Z 597.887,A -85,B 0,C 180,E1 -14328.927,E2 -14328.927} C_VEL
LIN {X 0,Y 349.868,Z 586.433,A -85,B 0,C 180,E1 -14329.737,E2 -14329.737} C_VEL
LIN {X 0,Y 350.199,Z 574.604,A -85,B 0,C 180,E1 -14330.362,E2 -14330.362} C_VEL
LIN {X 0,Y 350.34,Z 563.194,A -85,B 0,C 180,E1 -14330.769,E2 -14330.769} C_VEL
LIN {X 0,Y 350.663,Z 527.26,A -85,B 0,C 180,E1 -14331.543,E2 -14331.543} C_VEL
LIN {X 0,Y 351.049,Z 505.966,A -85,B 0,C 180,E1 -14331.98,E2 -14331.98} C_VEL
LIN {X 0,Y 341.041,Z 483.216,A -85,B 0,C 180,E1 -14333.225,E2 -14333.225} C_VEL
LIN {X 0,Y 340.82,Z 482.31,A -85,B 0,C 180,E1 -14333.387,E2 -14333.387} C_VEL
LIN {X 0,Y 340.757,Z 482.04,A -85,B 0,C 180,E1 -14334.361,E2 -14334.361} C_VEL
LIN {X 0,Y 340.779,Z 481.997,A -85,B 0,C 180,E1 -14337.425,E2 -14337.425} C_VEL
LIN {X 0,Y 340.094,Z 482.095,A -85,B 0,C 180,E1 -14338.41,E2 -14338.41} C_VEL
LIN {X 0,Y 337.221,Z 482.48,A -85,B 0,C 180,E1 -14340.013,E2 -14340.013} C_VEL
LIN {X 0,Y 334.788,Z 482.778,A -85,B 0,C 180,E1 -14341.311,E2 -14341.311} C_VEL
LIN {X 0,Y 333.732,Z 482.902,A -85,B 0,C 180,E1 -14342.315,E2 -14342.315} C_VEL
LIN {X 0,Y 333.64,Z 482.913,A -85,B 0,C 180,E1 -14342.656,E2 -14342.656} C_VEL
LIN {X 0,Y 333.675,Z 482.909,A -85,B 0,C 180,E1 -14346.138,E2 -14346.138} C_VEL
LIN {X 0,Y 333.645,Z 482.927,A -85,B 0,C 180,E1 -14349.191,E2 -14349.191} C_VEL
LIN {X 0,Y 333.63,Z 482.904,A -85,B 0,C 180,E1 -14352.499,E2 -14352.499} C_VEL
LIN {X 0,Y 333.619,Z 482.928,A -85,B 0,C 180,E1 -14355.958,E2 -14355.958} C_VEL
LIN {X 0,Y 333.643,Z 482.891,A -85,B 0,C 180,E1 -14359.315,E2 -14359.315} C_VEL
LIN {X 0,Y 333.661,Z 482.918,A -85,B 0,C 180,E1 -14363.167,E2 -14363.167} C_VEL
LIN {X 0,Y 333.669,Z 482.918,A -85,B 0,C 180,E1 -14365.341,E2 -14365.341} C_VEL
LIN {X 0,Y 333.697,Z 482.873,A -85,B 0,C 180,E1 -14369.71,E2 -14369.71} C_VEL
LIN {X 0,Y 333.739,Z 482.901,A -85,B 0,C 180,E1 -14372.401,E2 -14372.401} C_VEL
LIN {X 0,Y 333.721,Z 482.917,A -85,B 0,C 180,E1 -14375.09,E2 -14375.09} C_VEL
LIN {X 0,Y 333.668,Z 482.914,A -85,B 0,C 180,E1 -14379.018,E2 -14379.018} C_VEL
LIN {X 0,Y 333.787,Z 482.904,A -85,B 0,C 180,E1 -14381.589,E2 -14381.589} C_VEL
LIN {X 0,Y 333.801,Z 482.901,A -85,B 0,C 180,E1 -14385.576,E2 -14385.576} C_VEL
LIN {X 0,Y 333.826,Z 482.894,A -85,B 0,C 180,E1 -14389.078,E2 -14389.078} C_VEL
LIN {X 0,Y 334.017,Z 482.872,A -85,B 0,C 180,E1 -14392.747,E2 -14392.747} C_VEL
LIN {X 0,Y 333.805,Z 482.901,A -85,B 0,C 180,E1 -14395.169,E2 -14395.169} C_VEL
LIN {X 0,Y 334.099,Z 482.85,A -85,B 0,C 180,E1 -14397.589,E2 -14397.589} C_VEL
LIN {X 0,Y 334.26,Z 482.844,A -85,B 0,C 180,E1 -14400,E2 -14400} C_VEL
LIN {X 0,Y 334.1,Z 482.859,A -85,B 0,C 180,E1 -14402.411,E2 -14402.411} C_VEL
LIN {X 0,Y 334.011,Z 482.875,A -85,B 0,C 180,E1 -14406.039,E2 -14406.039} C_VEL
LIN {X 0,Y 333.951,Z 482.882,A -85,B 0,C 180,E1 -14408.471,E2 -14408.471} C_VEL
LIN {X 0,Y 333.784,Z 482.9,A -85,B 0,C 180,E1 -14412.155,E2 -14412.155} C_VEL
LIN {X 0,Y 333.77,Z 482.902,A -85,B 0,C 180,E1 -14415.887,E2 -14415.887} C_VEL
LIN {X 0,Y 333.788,Z 482.875,A -85,B 0,C 180,E1 -14418.654,E2 -14418.654} C_VEL
LIN {X 0,Y 333.656,Z 482.922,A -85,B 0,C 180,E1 -14422.281,E2 -14422.281} C_VEL
LIN {X 0,Y 333.73,Z 482.892,A -85,B 0,C 180,E1 -14426.247,E2 -14426.247} C_VEL
LIN {X 0,Y 333.706,Z 482.911,A -85,B 0,C 180,E1 -14428.973,E2 -14428.973} C_VEL
LIN {X 0,Y 333.638,Z 482.911,A -85,B 0,C 180,E1 -14432.588,E2 -14432.588} C_VEL
LIN {X 0,Y 333.671,Z 482.921,A -85,B 0,C 180,E1 -14436.14,E2 -14436.14} C_VEL
LIN {X 0,Y 333.643,Z 482.919,A -85,B 0,C 180,E1 -14439.193,E2 -14439.193} C_VEL
LIN {X 0,Y 333.63,Z 482.906,A -85,B 0,C 180,E1 -14442.501,E2 -14442.501} C_VEL
LIN {X 0,Y 333.666,Z 482.911,A -85,B 0,C 180,E1 -14445.968,E2 -14445.968} C_VEL
LIN {X 0,Y 333.699,Z 482.896,A -85,B 0,C 180,E1 -14449.305,E2 -14449.305} C_VEL
LIN {X 0,Y 333.733,Z 483.147,A -85,B 0,C 180,E1 -14452.964,E2 -14452.964} C_VEL
LIN {X 0,Y 337.149,Z 496.756,A -85,B 0,C 180,E1 -14456.2,E2 -14456.2} C_VEL
LIN {X 0,Y 340.149,Z 510.46,A -85,B 0,C 180,E1 -14459.246,E2 -14459.246} C_VEL
LIN {X 0,Y 340.353,Z 514.071,A -85,B 0,C 180,E1 -14459.986,E2 -14459.986} C_VEL
LIN {X 0,Y 337.67,Z 537.099,A -85,B 0,C 180,E1 -14464.414,E2 -14464.414} C_VEL
LIN {X 0,Y 336.847,Z 544.993,A -85,B 0,C 180,E1 -14465.911,E2 -14465.911} C_VEL
LIN {X 0,Y 339.598,Z 566.894,A -85,B 0,C 180,E1 -14466.64,E2 -14466.64} C_VEL
LIN {X 0,Y 342.918,Z 600.798,A -85,B 0,C 180,E1 -14467.617,E2 -14467.617} C_VEL
LIN {X 0,Y 341.828,Z 656.062,A -85,B 0,C 180,E1 -14468.794,E2 -14468.794} C_VEL
LIN {X 0,Y 341.16,Z 669.332,A -85,B 0,C 180,E1 -14469.304,E2 -14469.304} C_VEL
LIN {X 0,Y 339.898,Z 682.628,A -85,B 0,C 180,E1 -14470.053,E2 -14470.053} C_VEL
LIN {X 0,Y 338.677,Z 693.835,A -85,B 0,C 180,E1 -14470.924,E2 -14470.924} C_VEL
LIN {X 0,Y 337.197,Z 705.519,A -85,B 0,C 180,E1 -14472.096,E2 -14472.096} C_VEL
LIN {X 0,Y 335.976,Z 714.995,A -85,B 0,C 180,E1 -14473.285,E2 -14473.285} C_VEL
LIN {X 0,Y 334.773,Z 725.125,A -85,B 0,C 180,E1 -14474.849,E2 -14474.849} C_VEL
LIN {X 0,Y 333.783,Z 734.222,A -85,B 0,C 180,E1 -14476.608,E2 -14476.608} C_VEL
LIN {X 0,Y 333.068,Z 741.856,A -85,B 0,C 180,E1 -14478.437,E2 -14478.437} C_VEL
LIN {X 0,Y 332.715,Z 748.032,A -85,B 0,C 180,E1 -14480.271,E2 -14480.271} C_VEL
LIN {X 0,Y 332.659,Z 752.952,A -85,B 0,C 180,E1 -14482.107,E2 -14482.107} C_VEL
LIN {X 0,Y 332.752,Z 756.734,A -85,B 0,C 180,E1 -14483.938,E2 -14483.938} C_VEL
LIN {X 0,Y 332.939,Z 758.705,A -85,B 0,C 180,E1 -14485.157,E2 -14485.157} C_VEL
LIN {X 0,Y 333.076,Z 760.183,A -85,B 0,C 180,E1 -14486.371,E2 -14486.371} C_VEL
LIN {X 0,Y 333.507,Z 761.919,A -85,B 0,C 180,E1 -14488.793,E2 -14488.793} C_VEL
LIN {X 0,Y 333.63,Z 762.16,A -85,B 0,C 180,E1 -14490,E2 -14490} C_VEL
LIN {X 0,Y 333.507,Z 761.915,A -85,B 0,C 180,E1 -14491.207,E2 -14491.207} C_VEL
LIN {X 0,Y 333.079,Z 760.175,A -85,B 0,C 180,E1 -14493.629,E2 -14493.629} C_VEL
LIN {X 0,Y 332.943,Z 758.691,A -85,B 0,C 180,E1 -14494.843,E2 -14494.843} C_VEL
LIN {X 0,Y 332.717,Z 755.148,A -85,B 0,C 180,E1 -14496.886,E2 -14496.886} C_VEL
LIN {X 0,Y 332.67,Z 749.759,A -85,B 0,C 180,E1 -14499.116,E2 -14499.116} C_VEL
LIN {X 0,Y 332.863,Z 744.013,A -85,B 0,C 180,E1 -14500.954,E2 -14500.954} C_VEL
LIN {X 0,Y 333.463,Z 736.906,A -85,B 0,C 180,E1 -14502.785,E2 -14502.785} C_VEL
LIN {X 0,Y 334.269,Z 729.693,A -85,B 0,C 180,E1 -14504.302,E2 -14504.302} C_VEL
LIN {X 0,Y 335.323,Z 721.032,A -85,B 0,C 180,E1 -14505.811,E2 -14505.811} C_VEL
LIN {X 0,Y 336.46,Z 711.562,A -85,B 0,C 180,E1 -14507.16,E2 -14507.16} C_VEL
LIN {X 0,Y 337.94,Z 699.876,A -85,B 0,C 180,E1 -14508.49,E2 -14508.49} C_VEL
LIN {X 0,Y 339.341,Z 688.405,A -85,B 0,C 180,E1 -14509.509,E2 -14509.509} C_VEL
LIN {X 0,Y 340.51,Z 676.622,A -85,B 0,C 180,E1 -14510.304,E2 -14510.304} C_VEL
LIN {X 0,Y 341.476,Z 663.063,A -85,B 0,C 180,E1 -14510.952,E2 -14510.952} C_VEL
LIN {X 0,Y 341.952,Z 649.554,A -85,B 0,C 180,E1 -14511.356,E2 -14511.356} C_VEL
LIN {X 0,Y 342.875,Z 599.854,A -85,B 0,C 180,E1 -14512.39,E2 -14512.39} C_VEL
LIN {X 0,Y 339.23,Z 564.336,A -85,B 0,C 180,E1 -14513.425,E2 -14513.425} C_VEL
LIN {X 0,Y 336.837,Z 545.197,A -85,B 0,C 180,E1 -14514.05,E2 -14514.05} C_VEL
LIN {X 0,Y 339.142,Z 523.789,A -85,B 0,C 180,E1 -14518.127,E2 -14518.127} C_VEL
LIN {X 0,Y 340.366,Z 513.785,A -85,B 0,C 180,E1 -14520.046,E2 -14520.046} C_VEL
LIN {X 0,Y 340.091,Z 510.354,A -85,B 0,C 180,E1 -14520.76,E2 -14520.76} C_VEL
LIN {X 0,Y 337.352,Z 497.692,A -85,B 0,C 180,E1 -14523.559,E2 -14523.559} C_VEL
LIN {X 0,Y 334.152,Z 484.794,A -85,B 0,C 180,E1 -14526.591,E2 -14526.591} C_VEL
LIN {X 0,Y 333.696,Z 483.027,A -85,B 0,C 180,E1 -14527.076,E2 -14527.076} C_VEL
LIN {X 0,Y 333.696,Z 482.897,A -85,B 0,C 180,E1 -14530.759,E2 -14530.759} C_VEL
LIN {X 0,Y 333.666,Z 482.906,A -85,B 0,C 180,E1 -14534.263,E2 -14534.263} C_VEL
LIN {X 0,Y 333.639,Z 482.907,A -85,B 0,C 180,E1 -14537.618,E2 -14537.618} C_VEL
LIN {X 0,Y 333.648,Z 482.914,A -85,B 0,C 180,E1 -14541.201,E2 -14541.201} C_VEL
LIN {X 0,Y 333.671,Z 482.921,A -85,B 0,C 180,E1 -14543.86,E2 -14543.86} C_VEL
LIN {X 0,Y 333.638,Z 482.913,A -85,B 0,C 180,E1 -14547.412,E2 -14547.412} C_VEL
LIN {X 0,Y 333.706,Z 482.911,A -85,B 0,C 180,E1 -14551.027,E2 -14551.027} C_VEL
LIN {X 0,Y 333.73,Z 482.893,A -85,B 0,C 180,E1 -14553.753,E2 -14553.753} C_VEL
LIN {X 0,Y 333.656,Z 482.921,A -85,B 0,C 180,E1 -14557.719,E2 -14557.719} C_VEL
LIN {X 0,Y 333.786,Z 482.877,A -85,B 0,C 180,E1 -14561.589,E2 -14561.589} C_VEL
LIN {X 0,Y 333.801,Z 482.903,A -85,B 0,C 180,E1 -14565.576,E2 -14565.576} C_VEL
LIN {X 0,Y 333.826,Z 482.887,A -85,B 0,C 180,E1 -14569.078,E2 -14569.078} C_VEL
LIN {X 0,Y 334.001,Z 482.88,A -85,B 0,C 180,E1 -14572.747,E2 -14572.747} C_VEL
LIN {X 0,Y 333.806,Z 482.887,A -85,B 0,C 180,E1 -14575.169,E2 -14575.169} C_VEL
LIN {X 0,Y 334.1,Z 482.862,A -85,B 0,C 180,E1 -14577.589,E2 -14577.589} C_VEL
LIN {X 0,Y 334.26,Z 482.847,A -85,B 0,C 180,E1 -14580,E2 -14580} C_VEL
LIN {X 0,Y 334.1,Z 482.852,A -85,B 0,C 180,E1 -14582.411,E2 -14582.411} C_VEL
LIN {X 0,Y 333.988,Z 482.876,A -85,B 0,C 180,E1 -14586.599,E2 -14586.599} C_VEL
LIN {X 0,Y 333.843,Z 482.882,A -85,B 0,C 180,E1 -14589.696,E2 -14589.696} C_VEL
LIN {X 0,Y 333.789,Z 482.904,A -85,B 0,C 180,E1 -14593.392,E2 -14593.392} C_VEL
LIN {X 0,Y 333.739,Z 482.904,A -85,B 0,C 180,E1 -14597.147,E2 -14597.147} C_VEL
LIN {X 0,Y 333.726,Z 482.912,A -85,B 0,C 180,E1 -14599.691,E2 -14599.691} C_VEL
LIN {X 0,Y 333.668,Z 482.916,A -85,B 0,C 180,E1 -14603.591,E2 -14603.591} C_VEL
LIN {X 0,Y 333.73,Z 482.913,A -85,B 0,C 180,E1 -14606.247,E2 -14606.247} C_VEL
LIN {X 0,Y 333.706,Z 482.886,A -85,B 0,C 180,E1 -14608.973,E2 -14608.973} C_VEL
LIN {X 0,Y 333.638,Z 482.898,A -85,B 0,C 180,E1 -14612.588,E2 -14612.588} C_VEL
LIN {X 0,Y 333.672,Z 482.92,A -85,B 0,C 180,E1 -14616.14,E2 -14616.14} C_VEL
LIN {X 0,Y 333.642,Z 482.893,A -85,B 0,C 180,E1 -14619.193,E2 -14619.193} C_VEL
LIN {X 0,Y 333.63,Z 482.918,A -85,B 0,C 180,E1 -14622.501,E2 -14622.501} C_VEL
LIN {X 0,Y 333.617,Z 482.917,A -85,B 0,C 180,E1 -14625.96,E2 -14625.96} C_VEL
LIN {X 0,Y 333.645,Z 482.918,A -85,B 0,C 180,E1 -14629.316,E2 -14629.316} C_VEL
LIN {X 0,Y 333.664,Z 482.889,A -85,B 0,C 180,E1 -14633.169,E2 -14633.169} C_VEL
LIN {X 0,Y 333.673,Z 482.855,A -85,B 0,C 180,E1 -14635.342,E2 -14635.342} C_VEL
LIN {X 0,Y 333.704,Z 482.921,A -85,B 0,C 180,E1 -14639.711,E2 -14639.711} C_VEL
LIN {X 0,Y 333.739,Z 482.876,A -85,B 0,C 180,E1 -14642.402,E2 -14642.402} C_VEL
LIN {X 0,Y 333.746,Z 483.067,A -85,B 0,C 180,E1 -14646.169,E2 -14646.169} C_VEL
LIN {X 0,Y 334.027,Z 484.267,A -85,B 0,C 180,E1 -14646.378,E2 -14646.378} C_VEL
LIN {X 0,Y 344.246,Z 507.147,A -85,B 0,C 180,E1 -14647.676,E2 -14647.676} C_VEL
LIN {X 0,Y 344.503,Z 510.074,A -85,B 0,C 180,E1 -14647.76,E2 -14647.76} C_VEL
LIN {X 0,Y 343.738,Z 557.376,A -85,B 0,C 180,E1 -14648.755,E2 -14648.755} C_VEL
LIN {X 0,Y 343.674,Z 571.57,A -85,B 0,C 180,E1 -14649.17,E2 -14649.17} C_VEL
LIN {X 0,Y 343.214,Z 584.378,A -85,B 0,C 180,E1 -14649.785,E2 -14649.785} C_VEL
LIN {X 0,Y 342.555,Z 596.967,A -85,B 0,C 180,E1 -14650.643,E2 -14650.643} C_VEL
LIN {X 0,Y 341.656,Z 608.428,A -85,B 0,C 180,E1 -14651.678,E2 -14651.678} C_VEL
LIN {X 0,Y 340.674,Z 617.926,A -85,B 0,C 180,E1 -14652.75,E2 -14652.75} C_VEL
LIN {X 0,Y 339.552,Z 627.523,A -85,B 0,C 180,E1 -14654.083,E2 -14654.083} C_VEL
LIN {X 0,Y 338.488,Z 636.23,A -85,B 0,C 180,E1 -14655.573,E2 -14655.573} C_VEL
LIN {X 0,Y 337.402,Z 644.706,A -85,B 0,C 180,E1 -14657.367,E2 -14657.367} C_VEL
LIN {X 0,Y 336.358,Z 651.466,A -85,B 0,C 180,E1 -14659.161,E2 -14659.161} C_VEL
LIN {X 0,Y 335.678,Z 656.844,A -85,B 0,C 180,E1 -14660.966,E2 -14660.966} C_VEL
LIN {X 0,Y 334.856,Z 661.1,A -85,B 0,C 180,E1 -14662.766,E2 -14662.766} C_VEL
LIN {X 0,Y 334.515,Z 663.336,A -85,B 0,C 180,E1 -14663.97,E2 -14663.97} C_VEL
LIN {X 0,Y 334.212,Z 665.159,A -85,B 0,C 180,E1 -14665.175,E2 -14665.175} C_VEL
LIN {X 0,Y 334.155,Z 666.506,A -85,B 0,C 180,E1 -14666.383,E2 -14666.383} C_VEL
LIN {X 0,Y 333.986,Z 668.066,A -85,B 0,C 180,E1 -14668.794,E2 -14668.794} C_VEL
LIN {X 0,Y 333.961,Z 668.293,A -85,B 0,C 180,E1 -14670,E2 -14670} C_VEL
LIN {X 0,Y 333.985,Z 668.107,A -85,B 0,C 180,E1 -14671.206,E2 -14671.206} C_VEL
LIN {X 0,Y 334.151,Z 666.599,A -85,B 0,C 180,E1 -14673.618,E2 -14673.618} C_VEL
LIN {X 0,Y 334.201,Z 665.296,A -85,B 0,C 180,E1 -14674.825,E2 -14674.825} C_VEL
LIN {X 0,Y 334.718,Z 662.479,A -85,B 0,C 180,E1 -14676.631,E2 -14676.631} C_VEL
LIN {X 0,Y 335.436,Z 658.652,A -85,B 0,C 180,E1 -14678.433,E2 -14678.433} C_VEL
LIN {X 0,Y 336.072,Z 653.574,A -85,B 0,C 180,E1 -14680.299,E2 -14680.299} C_VEL
LIN {X 0,Y 336.991,Z 647.544,A -85,B 0,C 180,E1 -14682.037,E2 -14682.037} C_VEL
LIN {X 0,Y 338.127,Z 639.763,A -85,B 0,C 180,E1 -14683.829,E2 -14683.829} C_VEL
LIN {X 0,Y 339.287,Z 630.091,A -85,B 0,C 180,E1 -14685.621,E2 -14685.621} C_VEL
LIN {X 0,Y 340.351,Z 621.05,A -85,B 0,C 180,E1 -14686.958,E2 -14686.958} C_VEL
LIN {X 0,Y 341.497,Z 610.543,A -85,B 0,C 180,E1 -14688.205,E2 -14688.205} C_VEL
LIN {X 0,Y 342.463,Z 598.869,A -85,B 0,C 180,E1 -14689.308,E2 -14689.308} C_VEL
LIN {X 0,Y 343.254,Z 587.414,A -85,B 0,C 180,E1 -14690.134,E2 -14690.134} C_VEL
LIN {X 0,Y 343.639,Z 574.864,A -85,B 0,C 180,E1 -14690.8,E2 -14690.8} C_VEL
LIN {X 0,Y 343.768,Z 563.256,A -85,B 0,C 180,E1 -14691.209,E2 -14691.209} C_VEL
LIN {X 0,Y 344.089,Z 528.344,A -85,B 0,C 180,E1 -14691.973,E2 -14691.973} C_VEL
LIN {X 0,Y 344.526,Z 507.805,A -85,B 0,C 180,E1 -14692.399,E2 -14692.399} C_VEL
LIN {X 0,Y 334.681,Z 485.669,A -85,B 0,C 180,E1 -14693.639,E2 -14693.639} C_VEL
LIN {X 0,Y 333.819,Z 483.521,A -85,B 0,C 180,E1 -14693.825,E2 -14693.825} C_VEL
LIN {X 0,Y 333.738,Z 482.957,A -85,B 0,C 180,E1 -14694.079,E2 -14694.079} C_VEL
LIN {X 0,Y 333.716,Z 482.878,A -85,B 0,C 180,E1 -14697.808,E2 -14697.808} C_VEL
LIN {X 0,Y 333.69,Z 482.921,A -85,B 0,C 180,E1 -14700.362,E2 -14700.362} C_VEL
LIN {X 0,Y 333.64,Z 482.913,A -85,B 0,C 180,E1 -14702.656,E2 -14702.656} C_VEL
LIN {X 0,Y 332.955,Z 483.007,A -85,B 0,C 180,E1 -14703.662,E2 -14703.662} C_VEL
LIN {X 0,Y 330.102,Z 483.362,A -85,B 0,C 180,E1 -14705.301,E2 -14705.301} C_VEL
LIN {X 0,Y 327.701,Z 483.652,A -85,B 0,C 180,E1 -14706.628,E2 -14706.628} C_VEL
LIN {X 0,Y 326.68,Z 483.779,A -85,B 0,C 180,E1 -14707.655,E2 -14707.655} C_VEL
LIN {X 0,Y 326.601,Z 483.79,A -85,B 0,C 180,E1 -14708.003,E2 -14708.003} C_VEL
LIN {X 0,Y 326.574,Z 483.786,A -85,B 0,C 180,E1 -14711.845,E2 -14711.845} C_VEL
LIN {X 0,Y 326.554,Z 483.807,A -85,B 0,C 180,E1 -14715.251,E2 -14715.251} C_VEL
LIN {X 0,Y 326.574,Z 483.777,A -85,B 0,C 180,E1 -14718.868,E2 -14718.868} C_VEL
LIN {X 0,Y 326.623,Z 483.791,A -85,B 0,C 180,E1 -14722.761,E2 -14722.761} C_VEL
LIN {X 0,Y 326.602,Z 483.794,A -85,B 0,C 180,E1 -14725.98,E2 -14725.98} C_VEL
LIN {X 0,Y 326.655,Z 483.754,A -85,B 0,C 180,E1 -14730.34,E2 -14730.34} C_VEL
LIN {X 0,Y 326.684,Z 483.79,A -85,B 0,C 180,E1 -14734.516,E2 -14734.516} C_VEL
LIN {X 0,Y 326.615,Z 483.789,A -85,B 0,C 180,E1 -14738.543,E2 -14738.543} C_VEL
LIN {X 0,Y 326.738,Z 483.787,A -85,B 0,C 180,E1 -14741.177,E2 -14741.177} C_VEL
LIN {X 0,Y 326.756,Z 483.776,A -85,B 0,C 180,E1 -14745.433,E2 -14745.433} C_VEL
LIN {X 0,Y 326.762,Z 483.778,A -85,B 0,C 180,E1 -14748.839,E2 -14748.839} C_VEL
LIN {X 0,Y 326.968,Z 483.749,A -85,B 0,C 180,E1 -14752.59,E2 -14752.59} C_VEL
LIN {X 0,Y 326.772,Z 483.778,A -85,B 0,C 180,E1 -14755.065,E2 -14755.065} C_VEL
LIN {X 0,Y 327.04,Z 483.729,A -85,B 0,C 180,E1 -14757.537,E2 -14757.537} C_VEL
LIN {X 0,Y 327.21,Z 483.722,A -85,B 0,C 180,E1 -14760,E2 -14760} C_VEL
LIN {X 0,Y 327.041,Z 483.738,A -85,B 0,C 180,E1 -14762.463,E2 -14762.463} C_VEL
LIN {X 0,Y 326.985,Z 483.75,A -85,B 0,C 180,E1 -14766.169,E2 -14766.169} C_VEL
LIN {X 0,Y 326.798,Z 483.764,A -85,B 0,C 180,E1 -14769.907,E2 -14769.907} C_VEL
LIN {X 0,Y 326.752,Z 483.785,A -85,B 0,C 180,E1 -14773.686,E2 -14773.686} C_VEL
LIN {X 0,Y 326.691,Z 483.766,A -85,B 0,C 180,E1 -14777.528,E2 -14777.528} C_VEL
LIN {X 0,Y 326.649,Z 483.773,A -85,B 0,C 180,E1 -14780.136,E2 -14780.136} C_VEL
LIN {X 0,Y 326.645,Z 483.793,A -85,B 0,C 180,E1 -14784.129,E2 -14784.129} C_VEL
LIN {X 0,Y 326.679,Z 483.767,A -85,B 0,C 180,E1 -14786.858,E2 -14786.858} C_VEL
LIN {X 0,Y 326.634,Z 483.797,A -85,B 0,C 180,E1 -14790.612,E2 -14790.612} C_VEL
LIN {X 0,Y 326.602,Z 483.79,A -85,B 0,C 180,E1 -14794.02,E2 -14794.02} C_VEL
LIN {X 0,Y 326.623,Z 483.793,A -85,B 0,C 180,E1 -14797.239,E2 -14797.239} C_VEL
LIN {X 0,Y 326.575,Z 483.805,A -85,B 0,C 180,E1 -14801.132,E2 -14801.132} C_VEL
LIN {X 0,Y 326.578,Z 483.773,A -85,B 0,C 180,E1 -14804.753,E2 -14804.753} C_VEL
LIN {X 0,Y 326.62,Z 483.79,A -85,B 0,C 180,E1 -14808.162,E2 -14808.162} C_VEL
LIN {X 0,Y 326.642,Z 483.794,A -85,B 0,C 180,E1 -14812.134,E2 -14812.134} C_VEL
LIN {X 0,Y 326.685,Z 484.216,A -85,B 0,C 180,E1 -14812.506,E2 -14812.506} C_VEL
LIN {X 0,Y 330.156,Z 497.725,A -85,B 0,C 180,E1 -14815.815,E2 -14815.815} C_VEL
LIN {X 0,Y 333.106,Z 511.124,A -85,B 0,C 180,E1 -14818.876,E2 -14818.876} C_VEL
LIN {X 0,Y 333.48,Z 515.359,A -85,B 0,C 180,E1 -14819.776,E2 -14819.776} C_VEL
LIN {X 0,Y 330.739,Z 537.714,A -85,B 0,C 180,E1 -14824.176,E2 -14824.176} C_VEL
LIN {X 0,Y 330.068,Z 543.969,A -85,B 0,C 180,E1 -14825.384,E2 -14825.384} C_VEL
LIN {X 0,Y 333.227,Z 569.495,A -85,B 0,C 180,E1 -14826.247,E2 -14826.247} C_VEL
LIN {X 0,Y 336.289,Z 600.883,A -85,B 0,C 180,E1 -14827.175,E2 -14827.175} C_VEL
LIN {X 0,Y 335.203,Z 655.075,A -85,B 0,C 180,E1 -14828.354,E2 -14828.354} C_VEL
LIN {X 0,Y 334.527,Z 668.342,A -85,B 0,C 180,E1 -14828.874,E2 -14828.874} C_VEL
LIN {X 0,Y 333.368,Z 680.516,A -85,B 0,C 180,E1 -14829.564,E2 -14829.564} C_VEL
LIN {X 0,Y 331.947,Z 692.837,A -85,B 0,C 180,E1 -14830.522,E2 -14830.522} C_VEL
LIN {X 0,Y 330.427,Z 704.521,A -85,B 0,C 180,E1 -14831.717,E2 -14831.717} C_VEL
LIN {X 0,Y 329.192,Z 714.002,A -85,B 0,C 180,E1 -14832.93,E2 -14832.93} C_VEL
LIN {X 0,Y 327.894,Z 724.124,A -85,B 0,C 180,E1 -14834.523,E2 -14834.523} C_VEL
LIN {X 0,Y 327.145,Z 730.381,A -85,B 0,C 180,E1 -14835.718,E2 -14835.718} C_VEL
LIN {X 0,Y 326.254,Z 738.499,A -85,B 0,C 180,E1 -14837.56,E2 -14837.56} C_VEL
LIN {X 0,Y 325.713,Z 745.133,A -85,B 0,C 180,E1 -14839.432,E2 -14839.432} C_VEL
LIN {X 0,Y 325.571,Z 750.45,A -85,B 0,C 180,E1 -14841.309,E2 -14841.309} C_VEL
LIN {X 0,Y 325.62,Z 754.526,A -85,B 0,C 180,E1 -14843.14,E2 -14843.14} C_VEL
LIN {X 0,Y 325.861,Z 757.706,A -85,B 0,C 180,E1 -14845.051,E2 -14845.051} C_VEL
LIN {X 0,Y 326.029,Z 759.191,A -85,B 0,C 180,E1 -14846.292,E2 -14846.292} C_VEL
LIN {X 0,Y 326.447,Z 760.927,A -85,B 0,C 180,E1 -14848.766,E2 -14848.766} C_VEL
LIN {X 0,Y 326.603,Z 761.172,A -85,B 0,C 180,E1 -14850,E2 -14850} C_VEL
LIN {X 0,Y 326.447,Z 760.922,A -85,B 0,C 180,E1 -14851.234,E2 -14851.234} C_VEL
LIN {X 0,Y 326.032,Z 759.182,A -85,B 0,C 180,E1 -14853.708,E2 -14853.708} C_VEL
LIN {X 0,Y 325.864,Z 757.692,A -85,B 0,C 180,E1 -14854.949,E2 -14854.949} C_VEL
LIN {X 0,Y 325.648,Z 754.423,A -85,B 0,C 180,E1 -14856.901,E2 -14856.901} C_VEL
LIN {X 0,Y 325.571,Z 750.414,A -85,B 0,C 180,E1 -14858.691,E2 -14858.691} C_VEL
LIN {X 0,Y 325.762,Z 744.049,A -85,B 0,C 180,E1 -14860.881,E2 -14860.881} C_VEL
LIN {X 0,Y 326.367,Z 737.168,A -85,B 0,C 180,E1 -14862.751,E2 -14862.751} C_VEL
LIN {X 0,Y 327.172,Z 730.209,A -85,B 0,C 180,E1 -14864.302,E2 -14864.302} C_VEL
LIN {X 0,Y 328.192,Z 721.86,A -85,B 0,C 180,E1 -14865.844,E2 -14865.844} C_VEL
LIN {X 0,Y 329.27,Z 712.793,A -85,B 0,C 180,E1 -14867.226,E2 -14867.226} C_VEL
LIN {X 0,Y 330.846,Z 701.752,A -85,B 0,C 180,E1 -14868.58,E2 -14868.58} C_VEL
LIN {X 0,Y 332.151,Z 690.949,A -85,B 0,C 180,E1 -14869.627,E2 -14869.627} C_VEL
LIN {X 0,Y 333.603,Z 677.99,A -85,B 0,C 180,E1 -14870.582,E2 -14870.582} C_VEL
LIN {X 0,Y 334.7,Z 664.811,A -85,B 0,C 180,E1 -14871.276,E2 -14871.276} C_VEL
LIN {X 0,Y 335.255,Z 651.616,A -85,B 0,C 180,E1 -14871.723,E2 -14871.723} C_VEL
LIN {X 0,Y 336.269,Z 600.485,A -85,B 0,C 180,E1 -14872.817,E2 -14872.817} C_VEL
LIN {X 0,Y 332.591,Z 564.415,A -85,B 0,C 180,E1 -14873.896,E2 -14873.896} C_VEL
LIN {X 0,Y 330.022,Z 544.318,A -85,B 0,C 180,E1 -14874.567,E2 -14874.567} C_VEL
LIN {X 0,Y 330.493,Z 539.239,A -85,B 0,C 180,E1 -14875.506,E2 -14875.506} C_VEL
LIN {X 0,Y 332.895,Z 519.55,A -85,B 0,C 180,E1 -14879.377,E2 -14879.377} C_VEL
LIN {X 0,Y 333.523,Z 514.475,A -85,B 0,C 180,E1 -14880.379,E2 -14880.379} C_VEL
LIN {X 0,Y 331.977,Z 505.74,A -85,B 0,C 180,E1 -14882.312,E2 -14882.312} C_VEL
LIN {X 0,Y 328.623,Z 491.532,A -85,B 0,C 180,E1 -14885.642,E2 -14885.642} C_VEL
LIN {X 0,Y 326.655,Z 483.902,A -85,B 0,C 180,E1 -14887.589,E2 -14887.589} C_VEL
LIN {X 0,Y 326.626,Z 483.78,A -85,B 0,C 180,E1 -14891.141,E2 -14891.141} C_VEL
LIN {X 0,Y 326.587,Z 483.778,A -85,B 0,C 180,E1 -14894.753,E2 -14894.753} C_VEL
LIN {X 0,Y 326.573,Z 483.794,A -85,B 0,C 180,E1 -14898.154,E2 -14898.154} C_VEL
LIN {X 0,Y 326.594,Z 483.792,A -85,B 0,C 180,E1 -14901.387,E2 -14901.387} C_VEL
LIN {X 0,Y 326.614,Z 483.797,A -85,B 0,C 180,E1 -14904.851,E2 -14904.851} C_VEL
LIN {X 0,Y 326.602,Z 483.789,A -85,B 0,C 180,E1 -14907.455,E2 -14907.455} C_VEL
LIN {X 0,Y 326.656,Z 483.795,A -85,B 0,C 180,E1 -14910.34,E2 -14910.34} C_VEL
LIN {X 0,Y 326.684,Z 483.777,A -85,B 0,C 180,E1 -14914.516,E2 -14914.516} C_VEL
LIN {X 0,Y 326.614,Z 483.791,A -85,B 0,C 180,E1 -14918.543,E2 -14918.543} C_VEL
LIN {X 0,Y 326.738,Z 483.752,A -85,B 0,C 180,E1 -14921.177,E2 -14921.177} C_VEL
LIN {X 0,Y 326.756,Z 483.781,A -85,B 0,C 180,E1 -14925.433,E2 -14925.433} C_VEL
LIN {X 0,Y 326.762,Z 483.767,A -85,B 0,C 180,E1 -14928.839,E2 -14928.839} C_VEL
LIN {X 0,Y 326.953,Z 483.759,A -85,B 0,C 180,E1 -14932.59,E2 -14932.59} C_VEL
LIN {X 0,Y 326.773,Z 483.763,A -85,B 0,C 180,E1 -14935.065,E2 -14935.065} C_VEL
LIN {X 0,Y 327.041,Z 483.742,A -85,B 0,C 180,E1 -14937.537,E2 -14937.537} C_VEL
LIN {X 0,Y 327.21,Z 483.725,A -85,B 0,C 180,E1 -14940,E2 -14940} C_VEL
LIN {X 0,Y 327.041,Z 483.731,A -85,B 0,C 180,E1 -14942.463,E2 -14942.463} C_VEL
LIN {X 0,Y 326.957,Z 483.752,A -85,B 0,C 180,E1 -14946.589,E2 -14946.589} C_VEL
LIN {X 0,Y 326.798,Z 483.759,A -85,B 0,C 180,E1 -14949.907,E2 -14949.907} C_VEL
LIN {X 0,Y 326.752,Z 483.78,A -85,B 0,C 180,E1 -14953.686,E2 -14953.686} C_VEL
LIN {X 0,Y 326.692,Z 483.785,A -85,B 0,C 180,E1 -14957.528,E2 -14957.528} C_VEL
LIN {X 0,Y 326.652,Z 483.795,A -85,B 0,C 180,E1 -14960.136,E2 -14960.136} C_VEL
LIN {X 0,Y 326.645,Z 483.791,A -85,B 0,C 180,E1 -14964.13,E2 -14964.13} C_VEL
LIN {X 0,Y 326.68,Z 483.786,A -85,B 0,C 180,E1 -14966.858,E2 -14966.858} C_VEL
LIN {X 0,Y 326.634,Z 483.75,A -85,B 0,C 180,E1 -14970.612,E2 -14970.612} C_VEL
LIN {X 0,Y 326.602,Z 483.794,A -85,B 0,C 180,E1 -14974.02,E2 -14974.02} C_VEL
LIN {X 0,Y 326.623,Z 483.791,A -85,B 0,C 180,E1 -14977.239,E2 -14977.239} C_VEL
LIN {X 0,Y 326.574,Z 483.775,A -85,B 0,C 180,E1 -14981.132,E2 -14981.132} C_VEL
LIN {X 0,Y 326.554,Z 483.807,A -85,B 0,C 180,E1 -14984.749,E2 -14984.749} C_VEL
LIN {X 0,Y 326.574,Z 483.784,A -85,B 0,C 180,E1 -14988.155,E2 -14988.155} C_VEL
LIN {X 0,Y 326.622,Z 483.795,A -85,B 0,C 180,E1 -14991.392,E2 -14991.392} C_VEL
LIN {X 0,Y 326.618,Z 483.734,A -85,B 0,C 180,E1 -14994.852,E2 -14994.852} C_VEL
LIN {X 0,Y 326.607,Z 483.759,A -85,B 0,C 180,E1 -14997.456,E2 -14997.456} C_VEL
LIN {X 0,Y 326.661,Z 483.792,A -85,B 0,C 180,E1 -15000.342,E2 -15000.342} C_VEL
LIN {X 0,Y 326.691,Z 483.766,A -85,B 0,C 180,E1 -15004.517,E2 -15004.517} C_VEL
LIN {X 0,Y 326.729,Z 484.006,A -85,B 0,C 180,E1 -15005.646,E2 -15005.646} C_VEL
LIN {X 0,Y 327,Z 485.102,A -85,B 0,C 180,E1 -15005.831,E2 -15005.831} C_VEL
LIN {X 0,Y 337.184,Z 507.739,A -85,B 0,C 180,E1 -15007.171,E2 -15007.171} C_VEL
LIN {X 0,Y 337.985,Z 510.26,A -85,B 0,C 180,E1 -15007.288,E2 -15007.288} C_VEL
LIN {X 0,Y 337.203,Z 559.145,A -85,B 0,C 180,E1 -15008.34,E2 -15008.34} C_VEL
LIN {X 0,Y 337.088,Z 572.782,A -85,B 0,C 180,E1 -15008.752,E2 -15008.752} C_VEL
LIN {X 0,Y 336.627,Z 585.375,A -85,B 0,C 180,E1 -15009.372,E2 -15009.372} C_VEL
LIN {X 0,Y 335.933,Z 597.962,A -85,B 0,C 180,E1 -15010.246,E2 -15010.246} C_VEL
LIN {X 0,Y 334.997,Z 609.422,A -85,B 0,C 180,E1 -15011.301,E2 -15011.301} C_VEL
LIN {X 0,Y 333.967,Z 618.918,A -85,B 0,C 180,E1 -15012.392,E2 -15012.392} C_VEL
LIN {X 0,Y 332.798,Z 628.515,A -85,B 0,C 180,E1 -15013.751,E2 -15013.751} C_VEL
LIN {X 0,Y 331.686,Z 637.221,A -85,B 0,C 180,E1 -15015.27,E2 -15015.27} C_VEL
LIN {X 0,Y 330.548,Z 645.696,A -85,B 0,C 180,E1 -15017.1,E2 -15017.1} C_VEL
LIN {X 0,Y 329.458,Z 652.456,A -85,B 0,C 180,E1 -15018.931,E2 -15018.931} C_VEL
LIN {X 0,Y 328.739,Z 657.833,A -85,B 0,C 180,E1 -15020.774,E2 -15020.774} C_VEL
LIN {X 0,Y 327.886,Z 662.09,A -85,B 0,C 180,E1 -15022.611,E2 -15022.611} C_VEL
LIN {X 0,Y 327.525,Z 664.325,A -85,B 0,C 180,E1 -15023.841,E2 -15023.841} C_VEL
LIN {X 0,Y 327.207,Z 666.148,A -85,B 0,C 180,E1 -15025.071,E2 -15025.071} C_VEL
LIN {X 0,Y 327.141,Z 667.495,A -85,B 0,C 180,E1 -15026.305,E2 -15026.305} C_VEL
LIN {X 0,Y 326.963,Z 669.054,A -85,B 0,C 180,E1 -15028.768,E2 -15028.768} C_VEL
LIN {X 0,Y 326.934,Z 669.281,A -85,B 0,C 180,E1 -15030,E2 -15030} C_VEL
LIN {X 0,Y 326.961,Z 669.095,A -85,B 0,C 180,E1 -15031.232,E2 -15031.232} C_VEL
LIN {X 0,Y 327.136,Z 667.587,A -85,B 0,C 180,E1 -15033.695,E2 -15033.695} C_VEL
LIN {X 0,Y 327.195,Z 666.284,A -85,B 0,C 180,E1 -15034.929,E2 -15034.929} C_VEL
LIN {X 0,Y 327.738,Z 663.466,A -85,B 0,C 180,E1 -15036.773,E2 -15036.773} C_VEL
LIN {X 0,Y 328.485,Z 659.639,A -85,B 0,C 180,E1 -15038.613,E2 -15038.613} C_VEL
LIN {X 0,Y 329.159,Z 654.56,A -85,B 0,C 180,E1 -15040.518,E2 -15040.518} C_VEL
LIN {X 0,Y 330.121,Z 648.53,A -85,B 0,C 180,E1 -15042.292,E2 -15042.292} C_VEL
LIN {X 0,Y 331.307,Z 640.749,A -85,B 0,C 180,E1 -15044.119,E2 -15044.119} C_VEL
LIN {X 0,Y 332.523,Z 631.077,A -85,B 0,C 180,E1 -15045.947,E2 -15045.947} C_VEL
LIN {X 0,Y 333.633,Z 622.034,A -85,B 0,C 180,E1 -15047.31,E2 -15047.31} C_VEL
LIN {X 0,Y 334.829,Z 611.527,A -85,B 0,C 180,E1 -15048.581,E2 -15048.581} C_VEL
LIN {X 0,Y 335.814,Z 600.008,A -85,B 0,C 180,E1 -15049.692,E2 -15049.692} C_VEL
LIN {X 0,Y 336.647,Z 588.732,A -85,B 0,C 180,E1 -15050.523,E2 -15050.523} C_VEL
LIN {X 0,Y 337.049,Z 576.02,A -85,B 0,C 180,E1 -15051.218,E2 -15051.218} C_VEL
LIN {X 0,Y 337.197,Z 564.784,A -85,B 0,C 180,E1 -15051.628,E2 -15051.628} C_VEL
LIN {X 0,Y 337.552,Z 529.057,A -85,B 0,C 180,E1 -15052.428,E2 -15052.428} C_VEL
LIN {X 0,Y 337.982,Z 509.632,A -85,B 0,C 180,E1 -15052.837,E2 -15052.837} C_VEL
LIN {X 0,Y 328.699,Z 488.766,A -85,B 0,C 180,E1 -15054.045,E2 -15054.045} C_VEL
LIN {X 0,Y 326.81,Z 484.472,A -85,B 0,C 180,E1 -15054.359,E2 -15054.359} C_VEL
LIN {X 0,Y 326.703,Z 483.822,A -85,B 0,C 180,E1 -15054.632,E2 -15054.632} C_VEL
LIN {X 0,Y 326.65,Z 483.762,A -85,B 0,C 180,E1 -15058.25,E2 -15058.25} C_VEL
LIN {X 0,Y 326.589,Z 483.801,A -85,B 0,C 180,E1 -15061.095,E2 -15061.095} C_VEL
LIN {X 0,Y 326.606,Z 483.801,A -85,B 0,C 180,E1 -15064.019,E2 -15064.019} C_VEL
LIN {X 0,Y 326.601,Z 483.79,A -85,B 0,C 180,E1 -15068.003,E2 -15068.003} C_VEL
LIN {X 0,Y 325.958,Z 483.883,A -85,B 0,C 180,E1 -15069.032,E2 -15069.032} C_VEL
LIN {X 0,Y 323.156,Z 484.226,A -85,B 0,C 180,E1 -15070.709,E2 -15070.709} C_VEL
LIN {X 0,Y 320.743,Z 484.516,A -85,B 0,C 180,E1 -15072.066,E2 -15072.066} C_VEL
LIN {X 0,Y 319.664,Z 484.645,A -85,B 0,C 180,E1 -15073.117,E2 -15073.117} C_VEL
LIN {X 0,Y 319.553,Z 484.659,A -85,B 0,C 180,E1 -15073.473,E2 -15073.473} C_VEL
LIN {X 0,Y 319.558,Z 484.677,A -85,B 0,C 180,E1 -15077.017,E2 -15077.017} C_VEL
LIN {X 0,Y 319.542,Z 484.643,A -85,B 0,C 180,E1 -15080.37,E2 -15080.37} C_VEL
LIN {X 0,Y 319.575,Z 484.677,A -85,B 0,C 180,E1 -15084.456,E2 -15084.456} C_VEL
LIN {X 0,Y 319.527,Z 484.643,A -85,B 0,C 180,E1 -15088.137,E2 -15088.137} C_VEL
LIN {X 0,Y 319.611,Z 484.647,A -85,B 0,C 180,E1 -15091.588,E2 -15091.588} C_VEL
LIN {X 0,Y 319.599,Z 484.674,A -85,B 0,C 180,E1 -15095.303,E2 -15095.303} C_VEL
LIN {X 0,Y 319.597,Z 484.671,A -85,B 0,C 180,E1 -15099.4,E2 -15099.4} C_VEL
LIN {X 0,Y 319.651,Z 484.662,A -85,B 0,C 180,E1 -15102.073,E2 -15102.073} C_VEL
LIN {X 0,Y 319.725,Z 484.657,A -85,B 0,C 180,E1 -15106.007,E2 -15106.007} C_VEL
LIN {X 0,Y 319.751,Z 484.638,A -85,B 0,C 180,E1 -15109.873,E2 -15109.873} C_VEL
LIN {X 0,Y 319.926,Z 484.626,A -85,B 0,C 180,E1 -15112.426,E2 -15112.426} C_VEL
LIN {X 0,Y 319.741,Z 484.654,A -85,B 0,C 180,E1 -15114.956,E2 -15114.956} C_VEL
LIN {X 0,Y 319.984,Z 484.607,A -85,B 0,C 180,E1 -15117.482,E2 -15117.482} C_VEL
LIN {X 0,Y 320.162,Z 484.6,A -85,B 0,C 180,E1 -15120,E2 -15120} C_VEL
LIN {X 0,Y 319.984,Z 484.617,A -85,B 0,C 180,E1 -15122.518,E2 -15122.518} C_VEL
LIN {X 0,Y 319.939,Z 484.627,A -85,B 0,C 180,E1 -15126.306,E2 -15126.306} C_VEL
LIN {X 0,Y 319.83,Z 484.642,A -85,B 0,C 180,E1 -15128.848,E2 -15128.848} C_VEL
LIN {X 0,Y 319.674,Z 484.658,A -85,B 0,C 180,E1 -15132.7,E2 -15132.7} C_VEL
LIN {X 0,Y 319.693,Z 484.662,A -85,B 0,C 180,E1 -15135.296,E2 -15135.296} C_VEL
LIN {X 0,Y 319.645,Z 484.635,A -85,B 0,C 180,E1 -15139.257,E2 -15139.257} C_VEL
LIN {X 0,Y 319.557,Z 484.681,A -85,B 0,C 180,E1 -15143.32,E2 -15143.32} C_VEL
LIN {X 0,Y 319.629,Z 484.648,A -85,B 0,C 180,E1 -15146.089,E2 -15146.089} C_VEL
LIN {X 0,Y 319.585,Z 484.67,A -85,B 0,C 180,E1 -15148.934,E2 -15148.934} C_VEL
LIN {X 0,Y 319.527,Z 484.673,A -85,B 0,C 180,E1 -15151.862,E2 -15151.862} C_VEL
LIN {X 0,Y 319.575,Z 484.678,A -85,B 0,C 180,E1 -15155.544,E2 -15155.544} C_VEL
LIN {X 0,Y 319.554,Z 484.678,A -85,B 0,C 180,E1 -15159.669,E2 -15159.669} C_VEL
LIN {X 0,Y 319.56,Z 484.644,A -85,B 0,C 180,E1 -15163.469,E2 -15163.469} C_VEL
LIN {X 0,Y 319.601,Z 484.676,A -85,B 0,C 180,E1 -15167.026,E2 -15167.026} C_VEL
LIN {X 0,Y 319.62,Z 484.663,A -85,B 0,C 180,E1 -15171.196,E2 -15171.196} C_VEL
LIN {X 0,Y 319.625,Z 484.899,A -85,B 0,C 180,E1 -15171.925,E2 -15171.925} C_VEL
LIN {X 0,Y 323.035,Z 498.327,A -85,B 0,C 180,E1 -15175.319,E2 -15175.319} C_VEL
LIN {X 0,Y 326.397,Z 513.535,A -85,B 0,C 180,E1 -15178.885,E2 -15178.885} C_VEL
LIN {X 0,Y 326.651,Z 515.814,A -85,B 0,C 180,E1 -15179.386,E2 -15179.386} C_VEL
LIN {X 0,Y 324.192,Z 535.067,A -85,B 0,C 180,E1 -15183.268,E2 -15183.268} C_VEL
LIN {X 0,Y 323.298,Z 543.106,A -85,B 0,C 180,E1 -15184.851,E2 -15184.851} C_VEL
LIN {X 0,Y 327.566,Z 577.872,A -85,B 0,C 180,E1 -15186.026,E2 -15186.026} C_VEL
LIN {X 0,Y 329.754,Z 603.092,A -85,B 0,C 180,E1 -15186.77,E2 -15186.77} C_VEL
LIN {X 0,Y 328.592,Z 654.087,A -85,B 0,C 180,E1 -15187.896,E2 -15187.896} C_VEL
LIN {X 0,Y 327.902,Z 667.351,A -85,B 0,C 180,E1 -15188.426,E2 -15188.426} C_VEL
LIN {X 0,Y 326.709,Z 679.522,A -85,B 0,C 180,E1 -15189.128,E2 -15189.128} C_VEL
LIN {X 0,Y 325.245,Z 691.841,A -85,B 0,C 180,E1 -15190.103,E2 -15190.103} C_VEL
LIN {X 0,Y 323.644,Z 703.52,A -85,B 0,C 180,E1 -15191.319,E2 -15191.319} C_VEL
LIN {X 0,Y 322.218,Z 714.086,A -85,B 0,C 180,E1 -15192.712,E2 -15192.712} C_VEL
LIN {X 0,Y 321.064,Z 722.761,A -85,B 0,C 180,E1 -15194.121,E2 -15194.121} C_VEL
LIN {X 0,Y 320.1,Z 729.789,A -85,B 0,C 180,E1 -15195.486,E2 -15195.486} C_VEL
LIN {X 0,Y 319.257,Z 737.493,A -85,B 0,C 180,E1 -15197.283,E2 -15197.283} C_VEL
LIN {X 0,Y 318.657,Z 744.125,A -85,B 0,C 180,E1 -15199.195,E2 -15199.195} C_VEL
LIN {X 0,Y 318.5,Z 749.445,A -85,B 0,C 180,E1 -15201.115,E2 -15201.115} C_VEL
LIN {X 0,Y 318.55,Z 753.778,A -85,B 0,C 180,E1 -15203.128,E2 -15203.128} C_VEL
LIN {X 0,Y 318.786,Z 756.709,A -85,B 0,C 180,E1 -15204.941,E2 -15204.941} C_VEL
LIN {X 0,Y 318.98,Z 758.198,A -85,B 0,C 180,E1 -15206.21,E2 -15206.21} C_VEL
LIN {X 0,Y 319.387,Z 759.934,A -85,B 0,C 180,E1 -15208.739,E2 -15208.739} C_VEL
LIN {X 0,Y 319.574,Z 760.184,A -85,B 0,C 180,E1 -15210,E2 -15210} C_VEL
LIN {X 0,Y 319.388,Z 759.929,A -85,B 0,C 180,E1 -15211.261,E2 -15211.261} C_VEL
LIN {X 0,Y 318.983,Z 758.188,A -85,B 0,C 180,E1 -15213.79,E2 -15213.79} C_VEL
LIN {X 0,Y 318.79,Z 756.693,A -85,B 0,C 180,E1 -15215.059,E2 -15215.059} C_VEL
LIN {X 0,Y 318.587,Z 753.657,A -85,B 0,C 180,E1 -15216.928,E2 -15216.928} C_VEL
LIN {X 0,Y 318.5,Z 749.407,A -85,B 0,C 180,E1 -15218.885,E2 -15218.885} C_VEL
LIN {X 0,Y 318.751,Z 743.044,A -85,B 0,C 180,E1 -15221.123,E2 -15221.123} C_VEL
LIN {X 0,Y 319.353,Z 736.155,A -85,B 0,C 180,E1 -15223.036,E2 -15223.036} C_VEL
LIN {X 0,Y 320.159,Z 729.473,A -85,B 0,C 180,E1 -15224.562,E2 -15224.562} C_VEL
LIN {X 0,Y 321.328,Z 720.851,A -85,B 0,C 180,E1 -15226.192,E2 -15226.192} C_VEL
LIN {X 0,Y 322.516,Z 711.794,A -85,B 0,C 180,E1 -15227.598,E2 -15227.598} C_VEL
LIN {X 0,Y 324.063,Z 700.74,A -85,B 0,C 180,E1 -15228.984,E2 -15228.984} C_VEL
LIN {X 0,Y 325.695,Z 688.167,A -85,B 0,C 180,E1 -15230.197,E2 -15230.197} C_VEL
LIN {X 0,Y 327.088,Z 675.849,A -85,B 0,C 180,E1 -15231.094,E2 -15231.094} C_VEL
LIN {X 0,Y 328.126,Z 662.879,A -85,B 0,C 180,E1 -15231.765,E2 -15231.765} C_VEL
LIN {X 0,Y 328.7,Z 649.088,A -85,B 0,C 180,E1 -15232.22,E2 -15232.22} C_VEL
LIN {X 0,Y 329.616,Z 600.767,A -85,B 0,C 180,E1 -15233.274,E2 -15233.274} C_VEL
LIN {X 0,Y 326.159,Z 565.967,A -85,B 0,C 180,E1 -15234.337,E2 -15234.337} C_VEL
LIN {X 0,Y 323.293,Z 543.119,A -85,B 0,C 180,E1 -15235.127,E2 -15235.127} C_VEL
LIN {X 0,Y 325.875,Z 521.804,A -85,B 0,C 180,E1 -15239.382,E2 -15239.382} C_VEL
LIN {X 0,Y 326.575,Z 515.038,A -85,B 0,C 180,E1 -15240.755,E2 -15240.755} C_VEL
LIN {X 0,Y 324.104,Z 502.853,A -85,B 0,C 180,E1 -15243.569,E2 -15243.569} C_VEL
LIN {X 0,Y 321.166,Z 490.935,A -85,B 0,C 180,E1 -15246.485,E2 -15246.485} C_VEL
LIN {X 0,Y 319.631,Z 484.781,A -85,B 0,C 180,E1 -15248.099,E2 -15248.099} C_VEL
LIN {X 0,Y 319.594,Z 484.661,A -85,B 0,C 180,E1 -15251.611,E2 -15251.611} C_VEL
LIN {X 0,Y 319.536,Z 484.649,A -85,B 0,C 180,E1 -15255.265,E2 -15255.265} C_VEL
LIN {X 0,Y 319.525,Z 484.68,A -85,B 0,C 180,E1 -15258.711,E2 -15258.711} C_VEL
LIN {X 0,Y 319.55,Z 484.67,A -85,B 0,C 180,E1 -15262.349,E2 -15262.349} C_VEL
LIN {X 0,Y 319.555,Z 484.675,A -85,B 0,C 180,E1 -15265.123,E2 -15265.123} C_VEL
LIN {X 0,Y 319.565,Z 484.678,A -85,B 0,C 180,E1 -15269.057,E2 -15269.057} C_VEL
LIN {X 0,Y 319.603,Z 484.651,A -85,B 0,C 180,E1 -15272.498,E2 -15272.498} C_VEL
LIN {X 0,Y 319.599,Z 484.669,A -85,B 0,C 180,E1 -15275.303,E2 -15275.303} C_VEL
LIN {X 0,Y 319.594,Z 484.658,A -85,B 0,C 180,E1 -15279.4,E2 -15279.4} C_VEL
LIN {X 0,Y 319.651,Z 484.64,A -85,B 0,C 180,E1 -15282.073,E2 -15282.073} C_VEL
LIN {X 0,Y 319.725,Z 484.659,A -85,B 0,C 180,E1 -15286.007,E2 -15286.007} C_VEL
LIN {X 0,Y 319.745,Z 484.643,A -85,B 0,C 180,E1 -15289.872,E2 -15289.872} C_VEL
LIN {X 0,Y 319.907,Z 484.638,A -85,B 0,C 180,E1 -15292.426,E2 -15292.426} C_VEL
LIN {X 0,Y 319.742,Z 484.639,A -85,B 0,C 180,E1 -15294.956,E2 -15294.956} C_VEL
LIN {X 0,Y 319.984,Z 484.621,A -85,B 0,C 180,E1 -15297.482,E2 -15297.482} C_VEL
LIN {X 0,Y 320.162,Z 484.603,A -85,B 0,C 180,E1 -15300,E2 -15300} C_VEL
LIN {X 0,Y 319.985,Z 484.609,A -85,B 0,C 180,E1 -15302.518,E2 -15302.518} C_VEL
LIN {X 0,Y 319.92,Z 484.631,A -85,B 0,C 180,E1 -15306.575,E2 -15306.575} C_VEL
LIN {X 0,Y 319.745,Z 484.638,A -85,B 0,C 180,E1 -15310.128,E2 -15310.128} C_VEL
LIN {X 0,Y 319.724,Z 484.649,A -85,B 0,C 180,E1 -15314.724,E2 -15314.724} C_VEL
LIN {X 0,Y 319.683,Z 484.665,A -85,B 0,C 180,E1 -15319.038,E2 -15319.038} C_VEL
LIN {X 0,Y 319.557,Z 484.671,A -85,B 0,C 180,E1 -15323.321,E2 -15323.321} C_VEL
LIN {X 0,Y 319.629,Z 484.669,A -85,B 0,C 180,E1 -15326.089,E2 -15326.089} C_VEL
LIN {X 0,Y 319.584,Z 484.643,A -85,B 0,C 180,E1 -15328.934,E2 -15328.934} C_VEL
LIN {X 0,Y 319.527,Z 484.642,A -85,B 0,C 180,E1 -15331.863,E2 -15331.863} C_VEL
LIN {X 0,Y 319.576,Z 484.677,A -85,B 0,C 180,E1 -15335.544,E2 -15335.544} C_VEL
LIN {X 0,Y 319.555,Z 484.642,A -85,B 0,C 180,E1 -15339.67,E2 -15339.67} C_VEL
LIN {X 0,Y 319.555,Z 484.681,A -85,B 0,C 180,E1 -15343.468,E2 -15343.468} C_VEL
LIN {X 0,Y 319.558,Z 484.655,A -85,B 0,C 180,E1 -15347.018,E2 -15347.018} C_VEL
LIN {X 0,Y 319.545,Z 484.681,A -85,B 0,C 180,E1 -15350.372,E2 -15350.372} C_VEL
LIN {X 0,Y 319.557,Z 484.631,A -85,B 0,C 180,E1 -15353.573,E2 -15353.573} C_VEL
LIN {X 0,Y 319.576,Z 484.617,A -85,B 0,C 180,E1 -15356.687,E2 -15356.687} C_VEL
LIN {X 0,Y 319.592,Z 484.68,A -85,B 0,C 180,E1 -15359.618,E2 -15359.618} C_VEL
LIN {X 0,Y 319.606,Z 484.633,A -85,B 0,C 180,E1 -15362.499,E2 -15362.499} C_VEL
LIN {X 0,Y 319.698,Z 484.878,A -85,B 0,C 180,E1 -15365.064,E2 -15365.064} C_VEL
LIN {X 0,Y 319.982,Z 486.044,A -85,B 0,C 180,E1 -15365.263,E2 -15365.263} C_VEL
LIN {X 0,Y 329.42,Z 506.635,A -85,B 0,C 180,E1 -15366.547,E2 -15366.547} C_VEL
LIN {X 0,Y 331.394,Z 511.303,A -85,B 0,C 180,E1 -15366.811,E2 -15366.811} C_VEL
LIN {X 0,Y 330.628,Z 563.63,A -85,B 0,C 180,E1 -15367.973,E2 -15367.973} C_VEL
LIN {X 0,Y 330.42,Z 577.094,A -85,B 0,C 180,E1 -15368.452,E2 -15368.452} C_VEL
LIN {X 0,Y 329.92,Z 588.943,A -85,B 0,C 180,E1 -15369.096,E2 -15369.096} C_VEL
LIN {X 0,Y 329.126,Z 601.204,A -85,B 0,C 180,E1 -15370.023,E2 -15370.023} C_VEL
LIN {X 0,Y 328.201,Z 611.475,A -85,B 0,C 180,E1 -15371.021,E2 -15371.021} C_VEL
LIN {X 0,Y 326.971,Z 622.222,A -85,B 0,C 180,E1 -15372.326,E2 -15372.326} C_VEL
LIN {X 0,Y 325.809,Z 631.42,A -85,B 0,C 180,E1 -15373.715,E2 -15373.715} C_VEL
LIN {X 0,Y 324.726,Z 639.779,A -85,B 0,C 180,E1 -15375.268,E2 -15375.268} C_VEL
LIN {X 0,Y 323.495,Z 647.894,A -85,B 0,C 180,E1 -15377.134,E2 -15377.134} C_VEL
LIN {X 0,Y 322.321,Z 655.004,A -85,B 0,C 180,E1 -15379.189,E2 -15379.189} C_VEL
LIN {X 0,Y 321.564,Z 660.378,A -85,B 0,C 180,E1 -15381.2,E2 -15381.2} C_VEL
LIN {X 0,Y 320.766,Z 664.27,A -85,B 0,C 180,E1 -15383.079,E2 -15383.079} C_VEL
LIN {X 0,Y 320.203,Z 667.137,A -85,B 0,C 180,E1 -15384.963,E2 -15384.963} C_VEL
LIN {X 0,Y 320.127,Z 668.483,A -85,B 0,C 180,E1 -15386.224,E2 -15386.224} C_VEL
LIN {X 0,Y 319.94,Z 670.042,A -85,B 0,C 180,E1 -15388.741,E2 -15388.741} C_VEL
LIN {X 0,Y 319.908,Z 670.269,A -85,B 0,C 180,E1 -15390,E2 -15390} C_VEL
LIN {X 0,Y 319.937,Z 670.083,A -85,B 0,C 180,E1 -15391.259,E2 -15391.259} C_VEL
LIN {X 0,Y 320.122,Z 668.575,A -85,B 0,C 180,E1 -15393.776,E2 -15393.776} C_VEL
LIN {X 0,Y 320.191,Z 667.272,A -85,B 0,C 180,E1 -15395.037,E2 -15395.037} C_VEL
LIN {X 0,Y 320.76,Z 664.453,A -85,B 0,C 180,E1 -15396.921,E2 -15396.921} C_VEL
LIN {X 0,Y 321.538,Z 660.626,A -85,B 0,C 180,E1 -15398.801,E2 -15398.801} C_VEL
LIN {X 0,Y 322.252,Z 655.547,A -85,B 0,C 180,E1 -15400.746,E2 -15400.746} C_VEL
LIN {X 0,Y 323.257,Z 649.516,A -85,B 0,C 180,E1 -15402.557,E2 -15402.557} C_VEL
LIN {X 0,Y 324.495,Z 641.734,A -85,B 0,C 180,E1 -15404.422,E2 -15404.422} C_VEL
LIN {X 0,Y 325.769,Z 632.062,A -85,B 0,C 180,E1 -15406.287,E2 -15406.287} C_VEL
LIN {X 0,Y 326.928,Z 623.018,A -85,B 0,C 180,E1 -15407.676,E2 -15407.676} C_VEL
LIN {X 0,Y 328.166,Z 612.512,A -85,B 0,C 180,E1 -15408.973,E2 -15408.973} C_VEL
LIN {X 0,Y 329.229,Z 600.834,A -85,B 0,C 180,E1 -15410.117,E2 -15410.117} C_VEL
LIN {X 0,Y 330.1,Z 589.373,A -85,B 0,C 180,E1 -15410.973,E2 -15410.973} C_VEL
LIN {X 0,Y 330.481,Z 577.164,A -85,B 0,C 180,E1 -15411.653,E2 -15411.653} C_VEL
LIN {X 0,Y 330.677,Z 564.873,A -85,B 0,C 180,E1 -15412.101,E2 -15412.101} C_VEL
LIN {X 0,Y 331.066,Z 528.741,A -85,B 0,C 180,E1 -15412.921,E2 -15412.921} C_VEL
LIN {X 0,Y 331.479,Z 511.373,A -85,B 0,C 180,E1 -15413.293,E2 -15413.293} C_VEL
LIN {X 0,Y 322.178,Z 490.617,A -85,B 0,C 180,E1 -15414.542,E2 -15414.542} C_VEL
LIN {X 0,Y 319.839,Z 485.599,A -85,B 0,C 180,E1 -15414.895,E2 -15414.895} C_VEL
LIN {X 0,Y 319.649,Z 484.704,A -85,B 0,C 180,E1 -15415.17,E2 -15415.17} C_VEL
LIN {X 0,Y 319.579,Z 484.653,A -85,B 0,C 180,E1 -15418.934,E2 -15418.934} C_VEL
LIN {X 0,Y 319.53,Z 484.672,A -85,B 0,C 180,E1 -15421.861,E2 -15421.861} C_VEL
LIN {X 0,Y 319.579,Z 484.671,A -85,B 0,C 180,E1 -15425.542,E2 -15425.542} C_VEL
LIN {X 0,Y 319.556,Z 484.67,A -85,B 0,C 180,E1 -15428.009,E2 -15428.009} C_VEL
LIN {X 0,Y 319.523,Z 484.667,A -85,B 0,C 180,E1 -15431.596,E2 -15431.596} C_VEL
LIN {X 0,Y 319.553,Z 484.659,A -85,B 0,C 180,E1 -15433.473,E2 -15433.473} C_VEL
LIN {X 0,Y 318.817,Z 484.764,A -85,B 0,C 180,E1 -15434.523,E2 -15434.523} C_VEL
LIN {X 0,Y 315.923,Z 485.133,A -85,B 0,C 180,E1 -15436.233,E2 -15436.233} C_VEL
LIN {X 0,Y 313.531,Z 485.422,A -85,B 0,C 180,E1 -15437.62,E2 -15437.62} C_VEL
LIN {X 0,Y 312.538,Z 485.526,A -85,B 0,C 180,E1 -15438.693,E2 -15438.693} C_VEL
LIN {X 0,Y 312.473,Z 485.529,A -85,B 0,C 180,E1 -15439.056,E2 -15439.056} C_VEL
LIN {X 0,Y 312.516,Z 485.547,A -85,B 0,C 180,E1 -15442.613,E2 -15442.613} C_VEL
LIN {X 0,Y 312.515,Z 485.545,A -85,B 0,C 180,E1 -15446.31,E2 -15446.31} C_VEL
LIN {X 0,Y 312.54,Z 485.51,A -85,B 0,C 180,E1 -15450.349,E2 -15450.349} C_VEL
LIN {X 0,Y 312.597,Z 485.545,A -85,B 0,C 180,E1 -15454.064,E2 -15454.064} C_VEL
LIN {X 0,Y 312.561,Z 485.537,A -85,B 0,C 180,E1 -15457.527,E2 -15457.527} C_VEL
LIN {X 0,Y 312.632,Z 485.538,A -85,B 0,C 180,E1 -15461.656,E2 -15461.656} C_VEL
LIN {X 0,Y 312.687,Z 485.532,A -85,B 0,C 180,E1 -15465.686,E2 -15465.686} C_VEL
LIN {X 0,Y 312.695,Z 485.518,A -85,B 0,C 180,E1 -15469.642,E2 -15469.642} C_VEL
LIN {X 0,Y 312.865,Z 485.506,A -85,B 0,C 180,E1 -15472.254,E2 -15472.254} C_VEL
LIN {X 0,Y 312.711,Z 485.529,A -85,B 0,C 180,E1 -15474.842,E2 -15474.842} C_VEL
LIN {X 0,Y 312.985,Z 485.485,A -85,B 0,C 180,E1 -15478.713,E2 -15478.713} C_VEL
LIN {X 0,Y 313.113,Z 485.478,A -85,B 0,C 180,E1 -15480,E2 -15480} C_VEL
LIN {X 0,Y 312.931,Z 485.496,A -85,B 0,C 180,E1 -15482.574,E2 -15482.574} C_VEL
LIN {X 0,Y 312.896,Z 485.504,A -85,B 0,C 180,E1 -15486.448,E2 -15486.448} C_VEL
LIN {X 0,Y 312.76,Z 485.523,A -85,B 0,C 180,E1 -15489.05,E2 -15489.05} C_VEL
LIN {X 0,Y 312.627,Z 485.537,A -85,B 0,C 180,E1 -15492.991,E2 -15492.991} C_VEL
LIN {X 0,Y 312.631,Z 485.537,A -85,B 0,C 180,E1 -15495.65,E2 -15495.65} C_VEL
LIN {X 0,Y 312.602,Z 485.512,A -85,B 0,C 180,E1 -15499.225,E2 -15499.225} C_VEL
LIN {X 0,Y 312.523,Z 485.554,A -85,B 0,C 180,E1 -15502.782,E2 -15502.782} C_VEL
LIN {X 0,Y 312.597,Z 485.525,A -85,B 0,C 180,E1 -15505.936,E2 -15505.936} C_VEL
LIN {X 0,Y 312.54,Z 485.553,A -85,B 0,C 180,E1 -15509.651,E2 -15509.651} C_VEL
LIN {X 0,Y 312.514,Z 485.541,A -85,B 0,C 180,E1 -15513.689,E2 -15513.689} C_VEL
LIN {X 0,Y 312.516,Z 485.548,A -85,B 0,C 180,E1 -15517.387,E2 -15517.387} C_VEL
LIN {X 0,Y 312.486,Z 485.561,A -85,B 0,C 180,E1 -15520.71,E2 -15520.71} C_VEL
LIN {X 0,Y 312.482,Z 485.523,A -85,B 0,C 180,E1 -15524.204,E2 -15524.204} C_VEL
LIN {X 0,Y 312.546,Z 485.546,A -85,B 0,C 180,E1 -15527.906,E2 -15527.906} C_VEL
LIN {X 0,Y 312.594,Z 485.702,A -85,B 0,C 180,E1 -15531.341,E2 -15531.341} C_VEL
LIN {X 0,Y 315.823,Z 498.318,A -85,B 0,C 180,E1 -15534.651,E2 -15534.651} C_VEL
LIN {X 0,Y 319.271,Z 513.695,A -85,B 0,C 180,E1 -15538.377,E2 -15538.377} C_VEL
LIN {X 0,Y 319.755,Z 517.418,A -85,B 0,C 180,E1 -15539.225,E2 -15539.225} C_VEL
LIN {X 0,Y 317.282,Z 535.675,A -85,B 0,C 180,E1 -15542.994,E2 -15542.994} C_VEL
LIN {X 0,Y 316.55,Z 541.911,A -85,B 0,C 180,E1 -15544.259,E2 -15544.259} C_VEL
LIN {X 0,Y 319.704,Z 567.13,A -85,B 0,C 180,E1 -15545.169,E2 -15545.169} C_VEL
LIN {X 0,Y 322.602,Z 595.126,A -85,B 0,C 180,E1 -15546.061,E2 -15546.061} C_VEL
LIN {X 0,Y 323.172,Z 604.988,A -85,B 0,C 180,E1 -15546.336,E2 -15546.336} C_VEL
LIN {X 0,Y 322.004,Z 653.099,A -85,B 0,C 180,E1 -15547.419,E2 -15547.419} C_VEL
LIN {X 0,Y 321.27,Z 666.356,A -85,B 0,C 180,E1 -15547.957,E2 -15547.957} C_VEL
LIN {X 0,Y 320.041,Z 678.524,A -85,B 0,C 180,E1 -15548.673,E2 -15548.673} C_VEL
LIN {X 0,Y 318.55,Z 690.843,A -85,B 0,C 180,E1 -15549.667,E2 -15549.667} C_VEL
LIN {X 0,Y 316.884,Z 702.519,A -85,B 0,C 180,E1 -15550.906,E2 -15550.906} C_VEL
LIN {X 0,Y 315.382,Z 713.081,A -85,B 0,C 180,E1 -15552.325,E2 -15552.325} C_VEL
LIN {X 0,Y 314.2,Z 721.76,A -85,B 0,C 180,E1 -15553.764,E2 -15553.764} C_VEL
LIN {X 0,Y 313.043,Z 729.639,A -85,B 0,C 180,E1 -15555.339,E2 -15555.339} C_VEL
LIN {X 0,Y 312.136,Z 737.682,A -85,B 0,C 180,E1 -15557.319,E2 -15557.319} C_VEL
LIN {X 0,Y 311.522,Z 745.01,A -85,B 0,C 180,E1 -15559.602,E2 -15559.602} C_VEL
LIN {X 0,Y 311.439,Z 749.941,A -85,B 0,C 180,E1 -15561.566,E2 -15561.566} C_VEL
LIN {X 0,Y 311.551,Z 753.738,A -85,B 0,C 180,E1 -15563.524,E2 -15563.524} C_VEL
LIN {X 0,Y 311.699,Z 755.709,A -85,B 0,C 180,E1 -15564.826,E2 -15564.826} C_VEL
LIN {X 0,Y 311.93,Z 757.205,A -85,B 0,C 180,E1 -15566.124,E2 -15566.124} C_VEL
LIN {X 0,Y 312.329,Z 758.941,A -85,B 0,C 180,E1 -15568.711,E2 -15568.711} C_VEL
LIN {X 0,Y 312.545,Z 759.195,A -85,B 0,C 180,E1 -15570,E2 -15570} C_VEL
LIN {X 0,Y 312.33,Z 758.936,A -85,B 0,C 180,E1 -15571.289,E2 -15571.289} C_VEL
LIN {X 0,Y 311.933,Z 757.194,A -85,B 0,C 180,E1 -15573.876,E2 -15573.876} C_VEL
LIN {X 0,Y 311.704,Z 755.692,A -85,B 0,C 180,E1 -15575.174,E2 -15575.174} C_VEL
LIN {X 0,Y 311.533,Z 752.862,A -85,B 0,C 180,E1 -15576.967,E2 -15576.967} C_VEL
LIN {X 0,Y 311.426,Z 748.399,A -85,B 0,C 180,E1 -15579.089,E2 -15579.089} C_VEL
LIN {X 0,Y 311.726,Z 742.035,A -85,B 0,C 180,E1 -15581.377,E2 -15581.377} C_VEL
LIN {X 0,Y 312.36,Z 735.143,A -85,B 0,C 180,E1 -15583.333,E2 -15583.333} C_VEL
LIN {X 0,Y 313.142,Z 728.868,A -85,B 0,C 180,E1 -15584.806,E2 -15584.806} C_VEL
LIN {X 0,Y 314.468,Z 719.843,A -85,B 0,C 180,E1 -15586.555,E2 -15586.555} C_VEL
LIN {X 0,Y 315.553,Z 711.872,A -85,B 0,C 180,E1 -15587.832,E2 -15587.832} C_VEL
LIN {X 0,Y 317.137,Z 701.071,A -85,B 0,C 180,E1 -15589.247,E2 -15589.247} C_VEL
LIN {X 0,Y 318.552,Z 690.656,A -85,B 0,C 180,E1 -15590.333,E2 -15590.333} C_VEL
LIN {X 0,Y 320.066,Z 678.245,A -85,B 0,C 180,E1 -15591.326,E2 -15591.326} C_VEL
LIN {X 0,Y 321.302,Z 665.204,A -85,B 0,C 180,E1 -15592.083,E2 -15592.083} C_VEL
LIN {X 0,Y 321.993,Z 652.517,A -85,B 0,C 180,E1 -15592.582,E2 -15592.582} C_VEL
LIN {X 0,Y 323.074,Z 601.57,A -85,B 0,C 180,E1 -15593.73,E2 -15593.73} C_VEL
LIN {X 0,Y 319.702,Z 567.3,A -85,B 0,C 180,E1 -15594.805,E2 -15594.805} C_VEL
LIN {X 0,Y 316.533,Z 542.023,A -85,B 0,C 180,E1 -15595.707,E2 -15595.707} C_VEL
LIN {X 0,Y 319.04,Z 522.457,A -85,B 0,C 180,E1 -15599.711,E2 -15599.711} C_VEL
LIN {X 0,Y 319.691,Z 516.378,A -85,B 0,C 180,E1 -15600.978,E2 -15600.978} C_VEL
LIN {X 0,Y 317.427,Z 505.271,A -85,B 0,C 180,E1 -15603.607,E2 -15603.607} C_VEL
LIN {X 0,Y 314.397,Z 492.762,A -85,B 0,C 180,E1 -15606.74,E2 -15606.74} C_VEL
